// TwinCAT 3 PLC project TcBaseTest
// ProgramVersion: 3.1.4023.0
// libraries:
//   Tc2_Standard, * (Beckhoff Automation GmbH)
//   Tc2_System, * (Beckhoff Automation GmbH)
//   Tc2_Utilities, * (Beckhoff Automation GmbH)
//   Tc3_Module, * (Beckhoff Automation GmbH)
//   TcBase, * (TcBase)
//   TcUnit, * (www.tcunit.org)
// project tree:
//   Action Test/ FB_Action_Test.TcPOU, FB_ActivateAction.TcPOU
//   Collection Test/ FB_ListCapacity_Test.TcPOU, FB_List_proxy.TcPOU, FB_List_Test.TcPOU
//   Invocation Control Test/ FB_InvocationControlTestTask.TcPOU, FB_InvocationControl_Test.TcPOU
//   Object Test/ FB_Object_Test.TcPOU
//   Observer Pattern Test/ FB_ObserverPattern_Test.TcPOU, FB_Observer_LREAL_.TcPOU
//   / PlcTask.TcTTO
//   Programs/ Test.TcPOU
//   State Pattern Test/ FB_StatePattern_Test.TcPOU
//   State Pattern Test/Test Subjects/Dummy State Pattern/ FB_State1.TcPOU, FB_State2.TcPOU, FB_State3.TcPOU, FB_State4.TcPOU, FB_StateMachine1.TcPOU
//   State Pattern Test/Test Subjects/Season State Pattern/ E_Season.TcDUT, FB_Autumn.TcPOU, FB_Default.TcPOU, FB_SeasonBase.TcPOU, FB_SeasonStateMachine.TcPOU, FB_Spring.TcPOU, FB_Summer.TcPOU, FB_Winter.TcPOU, FB_Year.TcPOU, I_SeasonControl.TcIO, I_SeasonState.TcIO
//   Test Objects/ FB_ActionTestObject.TcPOU, FB_TestObject.TcPOU
// real-time tasks:
//   TASK PlcTask: cycle T#10ms, priority 20, ADS port 350

CONFIGURATION TcBaseTest
    RESOURCE PLC ON TwinCAT3
        TASK PlcTask(INTERVAL := T#10ms, PRIORITY := 20);
        PROGRAM Test WITH PlcTask : Test;
    END_RESOURCE
END_CONFIGURATION

// ---- State Pattern Test/Test Subjects/Season State Pattern/E_Season.TcDUT
{attribute 'qualified_only'}
{attribute 'strict'}
{attribute 'to_string'}
TYPE E_Season :
(
    Autumn,
    Winter,
    Spring,
    Summer
);
END_TYPE

// ---- State Pattern Test/Test Subjects/Season State Pattern/I_SeasonControl.TcIO
INTERFACE I_SeasonControl EXTENDS __SYSTEM.IQueryInterface

PROPERTY StateAutumn : I_State
GET
END_GET
END_PROPERTY

PROPERTY StateSpring : I_State
GET
END_GET
END_PROPERTY

PROPERTY StateSummer : I_State
GET
END_GET
END_PROPERTY

PROPERTY StateWinter : I_State
GET
END_GET
END_PROPERTY

END_INTERFACE

// ---- State Pattern Test/Test Subjects/Season State Pattern/I_SeasonState.TcIO
INTERFACE I_SeasonState EXTENDS I_State

PROPERTY bRaining : BOOL
GET
END_GET
END_PROPERTY

PROPERTY bSnowing : BOOL
GET
END_GET
END_PROPERTY

PROPERTY bSunShining : BOOL
GET
END_GET
END_PROPERTY

PROPERTY bWindBlowing : BOOL
GET
END_GET
END_PROPERTY

METHOD ChangeToSummerTyres
VAR_INPUT
END_VAR
END_METHOD

METHOD ChangeToWinterTyres
VAR_INPUT
END_VAR
END_METHOD

PROPERTY eState : E_Season
GET
END_GET
END_PROPERTY

METHOD ABSTRACT NextSeason
VAR_INPUT
END_VAR
END_METHOD

PROPERTY nLeavesState : BYTE
GET
END_GET
END_PROPERTY

PROPERTY nTyresType : BYTE
GET
END_GET
END_PROPERTY

PROPERTY sState : STRING(MAX_STRING_LENGTH)
GET
END_GET
END_PROPERTY

END_INTERFACE

// ---- Programs/Test.TcPOU
PROGRAM Test
VAR
    fbObjectTest: FB_Object_Test;
    fbListTest: FB_List_Test;
    fbListEnsureCapacityTest: FB_ListCapacity_Test;
    fbCallCtrlTest: FB_InvocationControl_Test;
    fbObserverPatternTest: FB_ObserverPattern_Test;
    fbStatePatternTest: FB_StatePattern_Test;
    fbActionTest: FB_Action_Test;
END_VAR

TcUnit.RUN();

END_PROGRAM

// ---- Object Test/FB_Object_Test.TcPOU
{attribute 'reflection'}
FUNCTION_BLOCK FB_Object_Test EXTENDS TcUnit.FB_TestSuite
VAR
    fbPathTester: FB_TestObject;
    _sTestPath: STRING(MAX_STRING_LENGTH) := CONCAT(_sPath, '.fbPathTester');

    {attribute 'instance-path'}
    {attribute 'noinit'}
    _sPath: STRING(MAX_STRING_LENGTH);
END_VAR

TestCompareObjectToSelfExpectTrue();
TestCompareTwoDifferentObjectsExpectFalse();
TestIdentityCorrectness();
TestPathCorrectness();

METHOD PRIVATE TestCompareObjectToSelfExpectTrue
VAR_INST
    fbObject1:      FB_TestObject;
END_VAR
TcUnit.TEST('TestCompareObjectToSelfExpectTrue');

THIS^.AssertTrue(Condition := fbObject1.Equals(fbObject1),
                 Message := 'Failed when comparing two equal objects');

TcUnit.TEST_FINISHED();
END_METHOD

METHOD PRIVATE TestCompareTwoDifferentObjectsExpectFalse
VAR_INST
    fbObject1:      FB_TestObject;
    fbObject2:      FB_TestObject;
END_VAR
TcUnit.TEST('TestCompareTwoDifferentObjectsExpectFalse');

THIS^.AssertFalse(Condition := fbObject1.Equals(fbObject2),
                  Message := 'Failed when comparing two equal objects');

TcUnit.TEST_FINISHED();
END_METHOD

METHOD PRIVATE TestIdentityCorrectness
VAR_INST
    fbObject: FB_TestObject;
END_VAR
TcUnit.TEST('TestIdentityCorrectness');

THIS^.AssertEquals_ULINT(Expected := ADR(fbObject),
                         Actual := fbObject.nIdentity,
                         Message := 'Object indentity is not true');

TcUnit.TEST_FINISHED();
END_METHOD

METHOD PRIVATE TestPathCorrectness
TcUnit.TEST('TestPathCorrectness');

THIS^.AssertEquals_STRING(Expected := THIS^._sTestPath,
                          Actual := THIS^.fbPathTester.sPath,
                          Message := 'Object path is not true');

TcUnit.TEST_FINISHED();
END_METHOD

END_FUNCTION_BLOCK

// ---- Test Objects/FB_TestObject.TcPOU
FUNCTION_BLOCK FB_TestObject EXTENDS FB_Object
VAR_INPUT
END_VAR
VAR_OUTPUT
END_VAR
VAR
    _nTest: INT;
END_VAR

PROPERTY nTest : INT
GET
nTest := THIS^._nTest;
END_GET
SET
THIS^._nTest := nTest;
END_SET
END_PROPERTY

END_FUNCTION_BLOCK

// ---- Collection Test/FB_List_Test.TcPOU
FUNCTION_BLOCK FB_List_Test EXTENDS TcUnit.FB_TestSuite
VAR
END_VAR

TestAdd5DifferentItemsExpectAll5Added();
TestAdd5TimesSameObjectExpectAll5Copies();
TestAddNullInterfaceExpectNothingAdded();
TestClearEmptyListExpectSuccess();
TestClearNonEmptyListExpectSuccess();
TestContainsAddedObjectsExpectSuccess();
TestContainsNullObjectExpectFailure();
TestContainsNullObjectFromEmptyListExpectFailure();
TestCopyToArrayOfCompatibleSizeExpectSuccess();
TestCopyToArrayOfIncompatibleSizeExpectFailure();
TestCopyToArrayWithInvalidIndexExpectFailure();
TestEmptyListMustHaveNoItem();
TestForEachWithActivateActionExpectSuccess();
TestForEachWithCylicTaskActionExpectSuccess();
TestIndexOfItem();
TestInsertIntoEmptyListExpectSuccess();
TestInsertIntoListOfItemsExpectSuccess();
TestLastIndexOfListOfMixedDuplicatesAndUniques();
TestRemoveByIndexAndReAddItemExpectCorrectItemOrder();
TestRemoveByIndexFromEmptyListExpectFailure();
TestRemoveByIndexFromListOf5DifferentItemsExpectSuccess();
TestRemoveByIndexFromListOf5ItemsExpectConsistentContents();
TestRemoveByInvalidIndexFromListOfItemsExpectFailure();
TestRemoveInvalidItemFromListExpectFailure();
TestRemoveValidItemFromListExpectSuccess();
{IF defined (LongTest)}
TestMeasureAddPerformanceWithVeryManyItemsAdded();
{END_IF}

METHOD PRIVATE TestAdd5DifferentItemsExpectAll5Added
VAR_INST
    fbList: FB_List_proxy(0);

    aObject: ARRAY [1..5] OF FB_TestObject;
    ipTmp: I_Object;
    ipCmp: I_Object;
    i: UDINT;
END_VAR
TcUnit.TEST('TestAdd5DifferentItemsExpectAll5Added');

FOR i := 1 TO SIZEOF(aObject)/SIZEOF(aObject[1]) DO
    THIS^.AssertEquals_DINT(Expected := TO_DINT(i - 1),
                            Actual := fbList.AddItem(aObject[i]),
                            Message := 'Failed to add object to list');
END_FOR

THIS^.AssertEquals_UDINT(Expected := SIZEOF(aObject)/SIZEOF(aObject[1]),
                         Actual := fbList.nCount,
                         Message := 'Unexpected number of items added to list');

FOR i := 1 TO SIZEOF(aObject)/SIZEOF(aObject[1]) DO
    ipTmp := fbList.ItemAt(TO_DINT(i - 1));
    ipCmp := aObject[i];
    THIS^.AssertTrue(Condition := ipTmp = ipCmp,
                     Message := CONCAT('Unexpected item at index ', TO_STRING(i)));
END_FOR

TcUnit.TEST_FINISHED();
END_METHOD

METHOD PRIVATE TestAdd5TimesSameObjectExpectAll5Copies
VAR_INST
    fbList: FB_List_proxy(0);

    nTimesToAdd: UDINT;
    fbObject: FB_TestObject;
    ipTmp: I_Object;
    ipCmp: I_Object;
    i: UDINT;
END_VAR
TcUnit.TEST('TestAdd5TimesSameObjectExpectAll5Copies');

nTimesToAdd := 5;

FOR i := 1 TO nTimesToAdd DO
    THIS^.AssertEquals_DINT(Expected := TO_DINT(i - 1),
                            Actual := fbList.AddItem(fbObject),
                            Message := 'Failed to add object to list');
END_FOR

THIS^.AssertEquals_UDINT(Expected := nTimesToAdd,
                         Actual := fbList.nCount,
                         Message := 'Unexpected number of items added to list');

FOR i := 1 TO nTimesToAdd DO
    ipTmp := fbList.ItemAt(TO_DINT(i - 1));
    ipCmp := fbObject;
    THIS^.AssertTrue(Condition := ipTmp = ipCmp,
                     Message := 'Unexpected item added to list');
END_FOR

TcUnit.TEST_FINISHED();
END_METHOD

METHOD PRIVATE TestAddNullInterfaceExpectNothingAdded
VAR_INST
    fbList: FB_List_proxy(0);

    ipTmp: I_Object;
    i: UDINT;
END_VAR
TcUnit.TEST('TestAddNullInterfaceExpectNothingAdded');

FOR i := 1 TO 5 DO
    THIS^.AssertEquals_DINT(Expected := -1,
                            Actual := fbList.AddItem(ipTmp),
                            Message := 'Null item added to list');
END_FOR

THIS^.AssertEquals_UDINT(Expected := 0,
                         Actual := fbList.nCount,
                         Message := 'List has item(s) in it, but it should not');

TcUnit.TEST_FINISHED();
END_METHOD

METHOD PRIVATE TestClearEmptyListExpectSuccess
VAR_INST
    fbList: FB_List_proxy(0);
END_VAR
TcUnit.TEST('TestClearEmptyListExpectSuccess');

fbList.Clear();

THIS^.AssertEquals_UDINT(Expected := 0,
                         Actual := fbList.nCount,
                         Message := 'List should be empty');

TcUnit.TEST_FINISHED();
END_METHOD

METHOD PRIVATE TestClearNonEmptyListExpectSuccess
VAR_INST
    fbList: FB_List_proxy(0);

    aObject: ARRAY [1..5] OF FB_TestObject;
    ipTmp: I_Object;
    i: UDINT;
END_VAR
TcUnit.TEST('TestClearNonEmptyListExpectSuccess');

FOR i := 1 TO SIZEOF(aObject)/SIZEOF(aObject[1]) DO
    fbList.AddItem(aObject[i]);
END_FOR

THIS^.AssertEquals_UDINT(Expected := SIZEOF(aObject)/SIZEOF(aObject[1]),
                         Actual := fbList.nCount,
                         Message := 'Unexpected number of items added to list');

fbList.Clear();

THIS^.AssertEquals_UDINT(Expected := 0,
                         Actual := fbList.nCount,
                         Message := 'List was not correctly cleared');

FOR i := 1 TO SIZEOF(aObject)/SIZEOF(aObject[1]) DO
    ipTmp := fbList.ItemAt(TO_DINT(i));
    THIS^.AssertTrue(Condition := ipTmp = 0,
                     Message := 'List was not correctly cleared');
END_FOR

TcUnit.TEST_FINISHED();
END_METHOD

METHOD PRIVATE TestContainsAddedObjectsExpectSuccess
VAR_INST
    fbList: FB_List_proxy(0);

    aObject: ARRAY [1..5] OF FB_TestObject;

    ipNull: I_Object;
    i: UDINT;
END_VAR
TcUnit.TEST('TestContainsAddedObjectsExpectSuccess');

FOR i := 1 TO SIZEOF(aObject)/SIZEOF(aObject[1]) DO
    fbList.AddItem(aObject[i]);
END_FOR

FOR i := 1 TO SIZEOF(aObject)/SIZEOF(aObject[1]) DO
    THIS^.AssertTrue(Condition := fbList.Contains(aObject[i]),
                     Message := 'List does not contain added item');
END_FOR

THIS^.AssertFalse(Condition := fbList.Contains(ipNull),
                  Message := 'List should not contain null object');

TcUnit.TEST_FINISHED();
END_METHOD

METHOD PRIVATE TestContainsNullObjectExpectFailure
VAR_INST
    fbList: FB_List_proxy(0);

    ipNull: I_Object;
END_VAR
TcUnit.TEST('TestContainsNullObjectExpectFailure');

THIS^.AssertFalse(Condition := fbList.Contains(ipNull),
                  Message := 'List should not contain null object');

TcUnit.TEST_FINISHED();
END_METHOD

METHOD PRIVATE TestContainsNullObjectFromEmptyListExpectFailure
VAR_INST
    fbList: FB_List_proxy(0);

    aObject: ARRAY [1..5] OF FB_TestObject;

    ipNull: I_Object;
    i: UDINT;
END_VAR
TcUnit.TEST('TestContainsNullObjectFromEmptyListExpectFailure');

FOR i := 1 TO SIZEOF(aObject)/SIZEOF(aObject[1]) DO
    fbList.AddItem(aObject[i]);
END_FOR

THIS^.AssertFalse(Condition := fbList.Contains(ipNull),
                  Message := 'List should not contain null object');

TcUnit.TEST_FINISHED();
END_METHOD

METHOD PRIVATE TestCopyToArrayOfCompatibleSizeExpectSuccess
VAR_INST
    fbList: FB_List_proxy(0);
    nObjectCount: UDINT;
    aSrcObject: ARRAY [1..10] OF FB_TestObject;
    aDestObject: ARRAY [1..10] OF I_Object;
    aDestObject2: ARRAY [1..30] OF I_Object;
    i: UDINT;
    ipObject: I_Object;

END_VAR
TcUnit.TEST('TestCopyToArrayOfCompatibleSizeExpectSuccess');

nObjectCount := SIZEOF(aSrcObject)/SIZEOF(aSrcObject[1]);
FOR i := 1 TO nObjectCount DO
    fbList.AddItem(aSrcObject[i]);
END_FOR

// Copy to same size array without offset
THIS^.AssertTrue(Condition := fbList.CopyToArray(aDestObject, 1),
                 Message := 'Failed to copy list to array of same size');

FOR i := 1 TO nObjectCount DO
    ipObject := aSrcObject[i];
    THIS^.AssertTrue(Condition := ipObject = aDestObject[i],
                     Message := 'Expected the same object after in array after copying from list');
END_FOR

// Copy to bigger array with offset
THIS^.AssertTrue(Condition := fbList.CopyToArray(aDestObject2, 14),
                 Message := 'Failed to copy list to array with bigger size');

FOR i := 1 TO nObjectCount DO
    ipObject := aSrcObject[i];
    THIS^.AssertTrue(Condition := ipObject = aDestObject2[i + 13],
                     Message := 'Expected the same object after in array after copying from list');
END_FOR

TcUnit.TEST_FINISHED();
END_METHOD

METHOD PRIVATE TestCopyToArrayOfIncompatibleSizeExpectFailure
VAR_INST
    fbList: FB_List_proxy(0);
    nObjectCount: UDINT;
    aSrcObject: ARRAY [1..10] OF FB_TestObject;
    aDestObject: ARRAY [1..5] OF I_Object;
    i: UDINT;
END_VAR
TcUnit.TEST('TestCopyToArrayOfIncompatibleSizeExpectFailure');

nObjectCount := SIZEOF(aSrcObject)/SIZEOF(aSrcObject[1]);
FOR i := 1 TO nObjectCount DO
    fbList.AddItem(aSrcObject[i]);
END_FOR

THIS^.AssertFalse(Condition := fbList.CopyToArray(aDestObject, 1),
                  Message := 'Failed to copy list to array of same size');

FOR i := 1 TO SIZEOF(aDestObject)/SIZEOF(aDestObject[1]) DO
    THIS^.AssertTrue(Condition := aDestObject[i] = 0,
                     Message := 'Array should be "empty" after copying due to being smaller than list');
END_FOR

TcUnit.TEST_FINISHED();
END_METHOD

METHOD PRIVATE TestCopyToArrayWithInvalidIndexExpectFailure
VAR_INST
    fbList: FB_List_proxy(0);
    nObjectCount: UDINT;
    aSrcObject: ARRAY [1..10] OF FB_TestObject;
    aDestObject: ARRAY [1..10] OF I_Object;
    aDestObject2: ARRAY [1..30] OF I_Object;
    i: UDINT;

END_VAR
TcUnit.TEST('TestCopyToArrayWithInvalidIndexExpectFailure');

nObjectCount := SIZEOF(aSrcObject)/SIZEOF(aSrcObject[1]);
FOR i := 1 TO nObjectCount DO
    fbList.AddItem(aSrcObject[i]);
END_FOR

// Copy to same size array
THIS^.AssertFalse(Condition := fbList.CopyToArray(aDestObject, 2),
                  Message := 'List should not copy items to array using invalid index');

FOR i := 1 TO nObjectCount DO
    THIS^.AssertTrue(Condition := 0 = aDestObject[i],
                     Message := 'Array should be "empty" after copying due to being smaller than list');
END_FOR

// Copy to bigger array
THIS^.AssertFalse(Condition := fbList.CopyToArray(aDestObject2, 22),
                  Message := 'List should not copy items to array using invalid index');

FOR i := 1 TO nObjectCount DO
    THIS^.AssertTrue(Condition := 0 = aDestObject2[i + 13],
                     Message := 'Array should be "empty" after copying due to being smaller than list');
END_FOR

THIS^.AssertFalse(Condition := fbList.CopyToArray(aDestObject2, 0),
                  Message := 'List should not copy items to array using invalid index');

FOR i := 1 TO nObjectCount DO
    THIS^.AssertTrue(Condition := 0 = aDestObject2[i + 13],
                     Message := 'Array should be "empty" after copying due to being smaller than list');
END_FOR

TcUnit.TEST_FINISHED();
END_METHOD

METHOD PRIVATE TestEmptyListMustHaveNoItem
VAR_INST
    fbList:     FB_List_proxy(0);
END_VAR
TcUnit.TEST('TestEmptyListMustHaveNoItem');

THIS^.AssertEquals_UDINT(Expected := 0,
                         Actual := fbList.nCount,
                         Message := 'Empty list must not have any item(s)');

TcUnit.TEST_FINISHED();
END_METHOD

METHOD PRIVATE TestForEachWithActivateActionExpectSuccess
VAR_INST
    i: UDINT;
    fbList: FB_List_proxy(0);
    aObject: ARRAY [1..10] OF FB_ActionTestObject;
    fbActivateObjects: FB_ActivateAction;
END_VAR
TcUnit.TEST('TestForEachWithActivateActionExpectSuccess');

FOR i := 1 TO SIZEOF(aObject)/SIZEOF(aObject[1]) DO
    fbList.AddItem(aObject[i]);
END_FOR

fbList.ForEach(fbActivateObjects.Inputs(TRUE));

FOR i := 1 TO SIZEOF(aObject)/SIZEOF(aObject[1]) DO
     THIS^.AssertTrue(Condition := aObject[1].bIsActivated,
                      Message := 'Failed to activate object(s)');
END_FOR

TcUnit.TEST_FINISHED();
END_METHOD

METHOD PRIVATE TestForEachWithCylicTaskActionExpectSuccess
VAR_INST
    nCyclesToRun: UDINT := 5;
    nCounter: UDINT := 0;
    i: UDINT;
    fbList: FB_List_proxy(0);
    aObject: ARRAY [1..10] OF FB_ActionTestObject;
    fbRunCyclicTask: FB_RunCyclicTasksAction;
END_VAR
TcUnit.TEST('TestForEachWithCylicTaskActionExpectSuccess');

IF nCounter = 0 THEN
    FOR i := 1 TO SIZEOF(aObject)/SIZEOF(aObject[1]) DO
        fbList.AddItem(aObject[i]);
    END_FOR
END_IF

fbList.ForEach(fbRunCyclicTask);
nCounter := nCounter + 1;

IF nCyclesToRun = nCounter THEN
    FOR i := 1 TO SIZEOF(aObject)/SIZEOF(aObject[1]) DO
        THIS^.AssertEquals_UDINT(Expected := nCyclesToRun,
                                 Actual := aObject[i].nCounter,
                                 Message := 'Unexpected counter value of cyclic object');
    END_FOR
    TcUnit.TEST_FINISHED();
END_IF
END_METHOD

METHOD PRIVATE TestIndexOfItem
VAR_INST
    fbList: FB_List_proxy(0);

    aObject: ARRAY [1..10] OF FB_TestObject;
    fbObject1: FB_TestObject;
    fbObject2: FB_TestObject;
    fbObject3: FB_TestObject;

    ipNull: I_Object;
    i: UDINT;
END_VAR
TcUnit.TEST('TestIndexQuerryCorrectness');

FOR i := 1 TO SIZEOF(aObject)/SIZEOF(aObject[1]) DO
    fbList.AddItem(aObject[i]);
END_FOR

FOR i := 1 TO SIZEOF(aObject)/SIZEOF(aObject[1]) DO
    THIS^.AssertEquals_DINT(Expected := TO_DINT(i - 1),
                            Actual := fbList.IndexOfItem(aObject[i]),
                            Message := 'Unexpected index of added item');
END_FOR

fbList.Clear();

FOR i := 1 TO SIZEOF(aObject)/SIZEOF(aObject[1]) DO
    THIS^.AssertEquals_DINT(Expected := -1,
                            Actual := fbList.IndexOfItem(aObject[i]),
                            Message := 'Item still found from list even though it has been cleared');
END_FOR

THIS^.AssertEquals_DINT(Expected := -1,
                        Actual := fbList.IndexOfItem(ipNull),
                        Message := 'Invalid result when querying index of a null item');

fbList.AddItem(fbObject1);
fbList.AddItem(fbObject3);
fbList.AddItem(fbObject1);
fbList.AddItem(fbObject2);
fbList.AddItem(fbObject2);

THIS^.AssertEquals_DINT(Expected := 0,
                        Actual := fbList.IndexOfItem(fbObject1),
                        Message := 'IndexOfItem() should return the index of the first match if there are multiple copies');
THIS^.AssertEquals_DINT(Expected := 1,
                        Actual := fbList.IndexOfItem(fbObject3),
                        Message := 'IndexOfItem() should return the index of the first match if there are multiple copies');
THIS^.AssertEquals_DINT(Expected := 3,
                        Actual := fbList.IndexOfItem(fbObject2),
                        Message := 'IndexOfItem() should return the index of the first match if there are multiple copies');


TcUnit.TEST_FINISHED();
END_METHOD

METHOD PRIVATE TestInsertIntoEmptyListExpectSuccess
VAR_INST
    fbList: FB_List_proxy(0);

    aObject: ARRAY [1..10] OF FB_TestObject;
    aInsPos: ARRAY [1..10] OF DINT;
    ipTmp: I_Object;
    ipCmp: I_Object;

    i: UDINT;
END_VAR
TcUnit.TEST('TestInsertIntoEmptyListExpectSuccess');

FOR i := 1 TO SIZEOF(aObject)/SIZEOF(aObject[1]) DO
    IF i = 4 THEN
        aInsPos[i] := 0;
    ELSIF i = 8 THEN
        aInsPos[i] := 4;;
    ELSIF i = 10 THEN
        aInsPos[i] := 1;
    ELSE
        aInsPos[i] := TO_DINT(i - 1);
    END_IF

    THIS^.AssertTrue(Condition := fbList.Insert(nIdx := aInsPos[i], aObject[i]),
                     Message := 'Could not insert item to list');

    ipTmp := fbList.ItemAt(aInsPos[i]);
    ipCmp := aObject[i];
    THIS^.AssertTrue(Condition := ipTmp = ipCmp,
                     Message := 'Added item is not at the expected index');
END_FOR

THIS^.AssertEquals_UDINT(Expected := SIZEOF(aObject)/SIZEOF(aObject[1]),
                         Actual := fbList.nCount,
                         Message := 'Unexpected number of items inserted to list');

FOR i := 1 TO SIZEOF(aObject)/SIZEOF(aObject[1]) DO
    THIS^.AssertTrue(Condition := fbList.Contains(aObject[i]),
                     Message := 'List does not contain inserted item');
END_FOR

TcUnit.TEST_FINISHED();
END_METHOD

METHOD PRIVATE TestInsertIntoListOfItemsExpectSuccess
VAR_INST
    fbList: FB_List_proxy(0);

    aObject: ARRAY [1..10] OF FB_TestObject;
    aObjectToInsert: ARRAY [1..3] OF FB_TestObject;
    aInsPos: ARRAY [1..3] OF DINT;
    ipTmp: I_Object;
    ipCmp: I_Object;

    i: UDINT;
END_VAR
TcUnit.TEST('TestInsertIntoListOfItemsExpectSuccess');

{region "Insert to head, end, and middle"}
FOR i := 1 TO SIZEOF(aObject)/SIZEOF(aObject[1]) DO
    fbList.AddItem(aObject[i]);
END_FOR

aInsPos[1] := 0;
aInsPos[2] := TO_DINT(fbList.nCount + 1);
aInsPos[3] := 3;

FOR i := 1 TO SIZEOF(aInsPos)/SIZEOF(aInsPos[1]) DO
    THIS^.AssertTrue(Condition := fbList.Insert(aInsPos[i], aObjectToInsert[i]),
                     Message := 'Failed to insert item into list');

    ipTmp := fbList.ItemAt(aInsPos[i]);
    ipCmp := aObjectToInsert[i];
    THIS^.AssertTrue(Condition := ipTmp = ipCmp,
                     Message := 'Added item is not at the expected index');
END_FOR

THIS^.AssertEquals_UDINT(Expected := SIZEOF(aObject)/SIZEOF(aObject[1])
                                     + SIZEOF(aObjectToInsert)/SIZEOF(aObjectToInsert[1]),
                         Actual := fbList.nCount,
                         Message := 'Unexpected number of items inserted to list');

FOR i := 1 TO SIZEOF(aObject)/SIZEOF(aObject[1]) DO
    THIS^.AssertTrue(Condition := fbList.Contains(aObject[i]),
                     Message := 'List does not contain inserted item');
END_FOR

FOR i := 1 TO SIZEOF(aObjectToInsert)/SIZEOF(aObjectToInsert[1]) DO
    THIS^.AssertTrue(Condition := fbList.Contains(aObjectToInsert[i]),
                     Message := 'List does not contain inserted item');
END_FOR
{endregion}

fbList.Clear();

{region "Insert to middle"}
FOR i := 1 TO SIZEOF(aObject)/SIZEOF(aObject[1]) DO
    fbList.AddItem(aObject[i]);
END_FOR

aInsPos[1] := 8;
aInsPos[2] := 5;
aInsPos[3] := 1;

FOR i := 1 TO SIZEOF(aInsPos)/SIZEOF(aInsPos[1]) DO
    THIS^.AssertTrue(Condition := fbList.Insert(aInsPos[i], aObjectToInsert[i]),
                     Message := 'Failed to insert item into list');

    ipTmp := fbList.ItemAt(aInsPos[i]);
    ipCmp := aObjectToInsert[i];
    THIS^.AssertTrue(Condition := ipTmp = ipCmp,
                     Message := 'Added item is not at the expected index');
END_FOR

THIS^.AssertEquals_UDINT(Expected := SIZEOF(aObject)/SIZEOF(aObject[1])
                                     + SIZEOF(aObjectToInsert)/SIZEOF(aObjectToInsert[1]),
                         Actual := fbList.nCount,
                         Message := 'Unexpected number of items inserted to list');

FOR i := 1 TO SIZEOF(aObject)/SIZEOF(aObject[1]) DO
    THIS^.AssertTrue(Condition := fbList.Contains(aObject[i]),
                     Message := 'List does not contain inserted item');
END_FOR

FOR i := 1 TO SIZEOF(aObjectToInsert)/SIZEOF(aObjectToInsert[1]) DO
    THIS^.AssertTrue(Condition := fbList.Contains(aObjectToInsert[i]),
                     Message := 'List does not contain inserted item');
END_FOR
{endregion}

TcUnit.TEST_FINISHED();
END_METHOD

METHOD PRIVATE TestLastIndexOfListOfMixedDuplicatesAndUniques
VAR_INST
    fbList: FB_List_proxy(0);

    aObject: ARRAY [1..5] OF FB_TestObject;
    aAddOrder: ARRAY[1..20] OF I_Object;
    aExpLastIdx: ARRAY [1..5] OF DINT;
    nIdx: UDINT;
    nObjectCount: UDINT;
    nTimesToAdd: UDINT;
    i: UDINT;
    fbRand: DRAND := (Seed := 128);
    sMessage: STRING(255);
END_VAR
TcUnit.TEST('TestLastIndexOfListOfMixedDuplicatesAndUniques');

nObjectCount := SIZEOF(aObject)/SIZEOF(aObject[1]);
nTimesToAdd := SIZEOF(aAddOrder)/SIZEOF(aAddOrder[1]);

FOR i := 1 TO nTimesToAdd DO
    fbRand();
    nIdx := TO_UDINT(fbRand.Num*(nObjectCount - 1)) + 1;
    aAddOrder[i] := aObject[nIdx];

    IF aExpLastIdx[nIdx] < TO_DINT(i) THEN
        aExpLastIdx[nIdx] := TO_DINT(i);
    END_IF
END_FOR

FOR i := 1 TO nTimesToAdd DO
    fbList.AddItem(aAddOrder[i]);
END_FOR

FOR i := 1 TO nObjectCount DO
    sMessage := Tc2_Standard.CONCAT('Unexpected last index of object at idx ', TO_STRING(i));
    THIS^.AssertEquals_DINT(Expected := aExpLastIdx[i] - 1,
                            Actual := fbList.LastIndexOf(aObject[i]),
                            Message := sMessage);
END_FOR

TcUnit.TEST_FINISHED();
END_METHOD

METHOD PRIVATE TestMeasureAddPerformanceWithVeryManyItemsAdded
VAR_INST
    fbList: FB_List_proxy(0);
    fbObject: FB_TestObject;
    fbProfiler: Tc2_Utilities.Profiler;

    nTimesToAdd: UDINT := 100000;
    i: UDINT;
    stProfileData: Tc2_Utilities.PROFILERSTRUCT;
    sMsg: STRING(255);
END_VAR
IF TcUnit.TEST_ORDERED('TestMeasureAddPerformanceWithVeryManyItemsAdded') THEN
    IF nTimesToAdd > 0 THEN
        fbProfiler(START := TRUE, RESET := TRUE);
        FOR i := 1 TO nTimesToAdd DO
            fbList.AddItem(fbObject);
        END_FOR

        THIS^.AssertEquals_UDINT(Expected := TO_UDINT(nTimesToAdd),
                                 Actual := fbList.nCount,
                                 Message := 'Unexpected number of items added to list');

        fbProfiler(START := FALSE);
        stProfileData := fbProfiler.DATA;

        sMsg := 'Took ';
        sMsg := CONCAT(sMsg, TO_STRING(stProfileData.LastExecTime));
        sMsg := CONCAT(sMsg, 'us to add ');
        sMsg := CONCAT(sMsg, TO_STRING(nTimesToAdd));
        sMsg := CONCAT(sMsg, ' item(s) to list. ');
        sMsg := CONCAT(sMsg, 'On average ');
        sMsg := CONCAT(sMsg, TO_STRING(fbProfiler.DATA.AverageExecTime/nTimesToAdd));
        sMsg := CONCAT(sMsg, 'us');
        sMsg := CONCAT(sMsg, ' per item');

        Tc2_System.ADSLOGSTR(msgCtrlMask := Tc2_System.ADSLOG_MSGTYPE_ERROR,
                             msgFmtStr := sMsg,
                             strArg := '');
    END_IF

    TcUnit.TEST_FINISHED();
END_IF
END_METHOD

METHOD PRIVATE TestRemoveByIndexAndReAddItemExpectCorrectItemOrder
VAR_INST
    fbList: FB_List_proxy(0);
    aObject: ARRAY [1..5] OF FB_TestObject;
    aIdx: ARRAY [1..5] OF UDINT
        := [3, 2, 4, 5, 1];
    nArraySize: UDINT;
    i: UDINT;
    j: UDINT;
END_VAR
TcUnit.TEST('TestRemoveByIndexAndReAddItemExpectCorrectItemOrder');
nArraySize := SIZEOF(aObject)/SIZEOF(aObject[1]);

FOR i := 1 TO nArraySize DO
    fbList.AddItem(aObject[i]);
END_FOR

FOR i := 1 TO nArraySize DO
    fbList.RemoveAt(fbList.IndexOfItem(aObject[aIdx[i]]));
    fbList.AddItem(aObject[aIdx[i]]);
END_FOR

FOR i := 1 TO nArraySize DO
    THIS^.AssertTrue(Condition := fbList.ItemAt(TO_DINT(i) - 1).Equals(aObject[aIdx[i]]),
                     Message := CONCAT('Unexpected item found at ', TO_STRING(i - 1)));
END_FOR

TcUnit.TEST_FINISHED();
END_METHOD

METHOD PRIVATE TestRemoveByIndexFromEmptyListExpectFailure
VAR_INST
    fbList: FB_List_proxy(0);

    aIdx: ARRAY[1..10] OF DINT := 
        [0, 1, 2, 3, 4, 5, 6, 7, 8, 9];

    i: UDINT;
END_VAR
TcUnit.TEST('TestRemoveByIndexFromEmptyListExpectFailure');

FOR i := 1 TO SIZEOF(aIdx)/SIZEOF(aIdx[1]) DO
    THIS^.AssertFalse(Condition := fbList.RemoveAt(aIdx[i]),
                      Message := 'Empty list should not have any item to be removed');
END_FOR

TcUnit.TEST_FINISHED();
END_METHOD

METHOD PRIVATE TestRemoveByIndexFromListOf5DifferentItemsExpectSuccess
VAR_INST
    fbList: FB_List_proxy(0);
    aObject: ARRAY [1..5] OF FB_TestObject;

    nArraySize: UDINT;
    i: UDINT;
END_VAR
TcUnit.TEST('TestRemoveItemFromListOf5DifferentItemsExpectSuccess');
nArraySize := SIZEOF(aObject)/SIZEOF(aObject[1]);

// Remove from last to first
FOR i := 1 TO nArraySize DO
    fbList.AddItem(aObject[i]);
END_FOR

FOR i := 1 TO nArraySize DO
    THIS^.AssertTrue(Condition := fbList.RemoveAt(TO_DINT(nArraySize - i)),
                     Message := 'Could not remove added item');

    THIS^.AssertEquals_UDINT(Expected := nArraySize - i,
                             Actual := fbList.nCount,
                             Message := 'Unexpected number of items after removal');
END_FOR

// Remove from first
FOR i := 1 TO nArraySize DO
    fbList.AddItem(aObject[i]);
END_FOR

FOR i := 1 TO nArraySize DO
    THIS^.AssertTrue(Condition := fbList.RemoveAt(0),
                     Message := 'Could not remove added item');

    THIS^.AssertEquals_UDINT(Expected := nArraySize - i,
                             Actual := fbList.nCount,
                             Message := 'Unexpected number of items after removal');
END_FOR

// Remove from middle to first
FOR i := 1 TO nArraySize DO
    fbList.AddItem(aObject[i]);
END_FOR

FOR i := 1 TO nArraySize DO
    THIS^.AssertTrue(Condition := fbList.RemoveAt(MAX(0, 3 - TO_DINT(i))),
                     Message := 'Could not remove added item');

    THIS^.AssertEquals_UDINT(Expected := nArraySize - i,
                             Actual := fbList.nCount,
                             Message := 'Unexpected number of items after removal');
END_FOR

TcUnit.TEST_FINISHED();
END_METHOD

METHOD PRIVATE TestRemoveByIndexFromListOf5ItemsExpectConsistentContents
VAR_INST
    fbList: FB_List_proxy(0);
    aObject: ARRAY [1..5] OF FB_TestObject;
    nArraySize: UDINT;
    i: UDINT;
    j: UDINT;
END_VAR
TcUnit.TEST('TestRemoveByIndexFromListOf5ItemsExpectConsistentContents');
nArraySize := SIZEOF(aObject)/SIZEOF(aObject[1]);

FOR i := 1 TO nArraySize DO
    fbList.AddItem(aObject[i]);
END_FOR

FOR i := 1 TO nArraySize DO
    fbList.RemoveAt(0);

    // After every removal, we check that the content of the list is correct
    IF fbList.nCount > 0 THEN
        FOR j := 0 TO fbList.nCount - 1 DO
            THIS^.AssertTrue(Condition := fbList.ItemAt(TO_DINT(j)).Equals(aObject[i + j + 1]),
                             Message := 'Unexpected list contents after removing item');
        END_FOR
    END_IF
END_FOR

TcUnit.TEST_FINISHED();
END_METHOD

METHOD PRIVATE TestRemoveByInvalidIndexFromListOfItemsExpectFailure
VAR_INST
    fbList: FB_List_proxy(0);

    aIdx: ARRAY[1..10] OF DINT := 
        [-1, 5, 6, 7, 10, -10, -3, -4, -2, 9];
    aObject: ARRAY [1..5] OF FB_TestObject;

    i: UDINT;
END_VAR
TcUnit.TEST('TestRemoveByInvalidIndexFromListOfItemsExpectFailure');

FOR i := 1 TO SIZEOF(aObject)/SIZEOF(aObject[1]) DO
    fbList.AddItem(aObject[i]);
END_FOR

FOR i := 1 TO SIZEOF(aIdx)/SIZEOF(aIdx[1]) DO
    THIS^.AssertFalse(Condition := fbList.RemoveAt(aIdx[i]),
                      Message := 'Removing item with out-of-bound index should not succeed');
END_FOR

THIS^.AssertEquals_UDINT(Expected := 5,
                         Actual := fbList.nCount,
                         Message := 'Item(s) were successfully removed from list with out-of-bound index');

TcUnit.TEST_FINISHED();
END_METHOD

METHOD PRIVATE TestRemoveInvalidItemFromListExpectFailure
VAR_INST
    fbList: FB_List_proxy(0);

    aObject: ARRAY [1..10] OF FB_TestObject;
    ipNull: I_Object;
    fbObject: FB_TestObject;

    i: UDINT;
END_VAR
TcUnit.TEST('TestRemoveInvalidItemFromListExpectFailure');

FOR i := 1 TO SIZEOF(aObject)/SIZEOF(aObject[1]) DO
    fbList.AddItem(aObject[i]);
END_FOR

THIS^.AssertFalse(Condition := fbList.Remove(ipNull),
                  Message := 'Unexpectedly removed a null item');

THIS^.AssertFalse(Condition := fbList.Remove(fbObject),
                  Message := 'List should not be able to remove item it does not contain');

THIS^.AssertEquals_UDINT(Expected := SIZEOF(aObject)/SIZEOF(aObject[1]),
                         Actual := fbList.nCount,
                         Message := 'Unexpected number of items after invalid removal');

FOR i := 1 TO SIZEOF(aObject)/SIZEOF(aObject[1]) DO
    THIS^.AssertTrue(Condition := fbList.Remove(aObject[i]),
                     Message := 'Could not remove added item');

    THIS^.AssertFalse(Condition := fbList.Remove(aObject[i]),
                      Message := 'Removed item was unexpectedly removed twice');

    THIS^.AssertEquals_UDINT(Expected := SIZEOF(aObject)/SIZEOF(aObject[1]) - i,
                             Actual := fbList.nCount,
                             Message := 'Unexpected number of items after removal');
END_FOR

TcUnit.TEST_FINISHED();
END_METHOD

METHOD PRIVATE TestRemoveValidItemFromListExpectSuccess
VAR_INST
    fbList: FB_List_proxy(0);

    aObject: ARRAY [1..10] OF FB_TestObject;

    i: UDINT;
END_VAR
TcUnit.TEST('TestRemoveValidItemFromListExpectSuccess');

FOR i := 1 TO SIZEOF(aObject)/SIZEOF(aObject[1]) DO
    fbList.AddItem(aObject[i]);
END_FOR

FOR i := 1 TO SIZEOF(aObject)/SIZEOF(aObject[1]) DO
    THIS^.AssertTrue(Condition := fbList.Remove(aObject[i]),
                     Message := 'Could not remove added item');

    THIS^.AssertEquals_UDINT(Expected := SIZEOF(aObject)/SIZEOF(aObject[1]) - i,
                             Actual := fbList.nCount,
                             Message := 'Unexpected number of items after removal');
END_FOR

TcUnit.TEST_FINISHED();
END_METHOD

END_FUNCTION_BLOCK

// ---- Collection Test/FB_List_proxy.TcPOU
FUNCTION_BLOCK FB_List_proxy EXTENDS TcBase.FB_List
VAR_INPUT
END_VAR
VAR_OUTPUT
END_VAR
VAR
END_VAR

END_FUNCTION_BLOCK

// ---- Test Objects/FB_ActionTestObject.TcPOU
FUNCTION_BLOCK FB_ActionTestObject EXTENDS TcBase.FB_Object IMPLEMENTS TcBase.I_CyclicTask
VAR
    _nCounter: UDINT;
    _bActivated: BOOL;
END_VAR

METHOD Activate
VAR_INPUT
    bActivate: BOOL;
END_VAR
THIS^._bActivated := bActivate;
END_METHOD

PROPERTY bIsActivated : BOOL
GET
bIsActivated := THIS^._bActivated;
END_GET
END_PROPERTY

PROPERTY nCounter : UDINT
GET
nCounter := THIS^._nCounter;
END_GET
END_PROPERTY

METHOD Run
VAR_INPUT
END_VAR
THIS^._nCounter := THIS^._nCounter + 1;
END_METHOD

END_FUNCTION_BLOCK

// ---- Action Test/FB_ActivateAction.TcPOU
FUNCTION_BLOCK FB_ActivateAction EXTENDS TcBase.FB_Action
VAR
    _bActivated: BOOL;
END_VAR

METHOD  Execute
VAR_INPUT
    ipObject: I_Object;
END_VAR
VAR
    p: POINTER TO FB_ActionTestObject;
END_VAR
__QUERYPOINTER(ipObject, p);

IF p <> 0 THEN
    p^.Activate(THIS^._bActivated);
END_IF
END_METHOD

METHOD Inputs : TcBase.I_Action
VAR_INPUT
    bActivate: BOOL;
END_VAR
Inputs := THIS^;
THIS^._bActivated := bActivate;
END_METHOD

END_FUNCTION_BLOCK

// ---- Collection Test/FB_ListCapacity_Test.TcPOU
FUNCTION_BLOCK FB_ListCapacity_Test EXTENDS TcUnit.FB_TestSuite
VAR_INPUT
END_VAR
VAR_OUTPUT
END_VAR
VAR
END_VAR

TestInitializeCapacityWithNonZeroValuesExpectSuccess();

METHOD PRIVATE TestInitializeCapacityWithNonZeroValuesExpectSuccess
VAR_INST
    aList: ARRAY [1..5] OF FB_List[(4), (10), (20), (100), (1000)];
    aExpected: ARRAY [1..5] OF UDINT := [4, 10, 20, 100, 1000];
    i: UDINT;
END_VAR
TcUnit.TEST('TestInitializeCapacityWithNonZeroValuesExpectSuccess');

FOR i := 1 TO SIZEOF(aList)/SIZEOF(aList[1]) DO
    THIS^.AssertEquals_UDINT(Expected := aExpected[i],
                             Actual := aList[i].nCapacity,
                             Message := 'Unexpected capacity');
END_FOR

TcUnit.TEST_FINISHED();
END_METHOD

END_FUNCTION_BLOCK

// ---- Invocation Control Test/FB_InvocationControl_Test.TcPOU
FUNCTION_BLOCK FB_InvocationControl_Test EXTENDS TcUnit.FB_TestSuite
VAR
    
END_VAR

RunAllTheTimeExpectCalledCyclicallyTrue();
RunAllTheTimeExpectNewInvocationOnce();
RunOnceExpectNewInvocationOnce();
RunOncePerCycleExpectMultipleCallAlwaysFalse();
RunThricePerCycleExpectMultipleCallTrue();

METHOD PRIVATE RunAllTheTimeExpectCalledCyclicallyTrue
VAR_INST
    fbCallCtrl:             FB_InvocationControl;
    fbCallCtrlTestTask:     FB_InvocationControlTestTask;
END_VAR
TcUnit.TEST('RunAllTheTimeExpectCalledCyclicallyTrue');

fbCallCtrlTestTask.SetRunCondition(5).Run();

IF fbCallCtrlTestTask.nCycleCounter = 1 THEN
    THIS^.AssertFalse(Condition := fbCallCtrl.bCalledCyclically,
                      Message := '$'bCalledCyclically$' should be false as Track() has not been called at all');
END_IF

fbCallCtrl.Track();

THIS^.AssertTrue(Condition := fbCallCtrl.bCalledCyclically,
                 Message := '$'bCalledCyclically$' is false, but it should be true');

THIS^.AssertTrue(Condition := fbCallCtrl.bCalledThisCycle,
                 Message := '$'bCalledThisCycle$' is false, but it should be true');

IF fbCallCtrlTestTask.nCycleCounter > 1 THEN
    THIS^.AssertTrue(Condition := fbCallCtrl.bCalledLastCycle,
                     Message := '$'bCalledLastCycle$' is false, but it should be true');
    IF NOT fbCallCtrl.bCalledLastCycle THEN
        ADSLOGSTR(msgCtrlMask := ADSLOG_MSGTYPE_ERROR,
                  msgFmtStr := fbCallCtrl.ToString(),
                  strArg := '');
    END_IF
ELSE
    THIS^.AssertFalse(Condition := fbCallCtrl.bCalledLastCycle,
                      Message := '$'bCalledLastCycle$' should not be true on the first cycle it is called');
END_IF

IF fbCallCtrlTestTask.bDone THEN
    TcUnit.TEST_FINISHED();
END_IF
END_METHOD

METHOD PRIVATE RunAllTheTimeExpectNewInvocationOnce
VAR_INST
    fbCallCtrl:             FB_InvocationControl;
    fbCallCtrlTestTask:     FB_InvocationControlTestTask;
END_VAR
TcUnit.TEST('RunAllTheTimeExpectNewInvocationOnce');

fbCallCtrlTestTask.SetRunCondition(5).Run();

fbCallCtrl.Track();

IF fbCallCtrlTestTask.nCycleCounter = 1 THEN
    THIS^.AssertTrue(Condition := fbCallCtrl.bNewInvocation,
                     Message := '$'bNewInvocation$' is false, but it should be true');
ELSE
    THIS^.Assertfalse(Condition := fbCallCtrl.bNewInvocation,
                      Message := '$'bNewInvocation$' is true, but it should be false');
END_IF

IF fbCallCtrlTestTask.bDone THEN
    TcUnit.TEST_FINISHED();
END_IF
END_METHOD

METHOD PRIVATE RunOnceExpectNewInvocationOnce
VAR_INST
    fbCallCtrl:             FB_InvocationControl;
    fbCallCtrlTestTask:     FB_InvocationControlTestTask;
END_VAR
TcUnit.TEST('RunOnceExpectNewInvocationOnce');

fbCallCtrlTestTask.SetRunCondition(5).Run();

IF fbCallCtrlTestTask.nCycleCounter = 3 THEN
    fbCallCtrl.Track();
    THIS^.AssertTrue(Condition := fbCallCtrl.bNewInvocation,
                     Message := '$'bNewInvocation$' is false, but it should be true');
ELSE
    THIS^.AssertFalse(Condition := fbCallCtrl.bNewInvocation,
                      Message := '$'bNewInvocation$' is trie, but it should be false');
END_IF

IF fbCallCtrlTestTask.bDone THEN
    TcUnit.TEST_FINISHED();
END_IF
END_METHOD

METHOD PRIVATE RunOncePerCycleExpectMultipleCallAlwaysFalse
VAR_INST
    fbCallCtrl:             FB_InvocationControl;
    fbCallCtrlTestTask:     FB_InvocationControlTestTask;
END_VAR
TcUnit.TEST('RunOncePerCycleExpectMultipleCallAlwaysFalse');

fbCallCtrlTestTask.SetRunCondition(5).Run();

THIS^.AssertFalse(Condition := fbCallCtrl.bMultipleCall,
                  Message := '$'bMultipleCall$' is true, but it should be false');

fbCallCtrl.Track();

THIS^.AssertFalse(Condition := fbCallCtrl.bMultipleCall,
                  Message := '$'bMultipleCall$' is true, but it should be false');


IF fbCallCtrlTestTask.bDone THEN
    TcUnit.TEST_FINISHED();
END_IF
END_METHOD

METHOD PRIVATE RunThricePerCycleExpectMultipleCallTrue
VAR_INST
    fbCallCtrl:             FB_InvocationControl;
    fbCallCtrlTestTask:     FB_InvocationControlTestTask;
END_VAR
TcUnit.TEST('RunThricePerCycleExpectMultipleCallTrue');

fbCallCtrlTestTask.SetRunCondition(5).Run();

IF fbCallCtrlTestTask.nCycleCounter > 1 THEN
    THIS^.AssertTrue(Condition := fbCallCtrl.bMultipleCall,
                     Message := '$'bMultipleCall$' is false, but it should be true');
END_IF

fbCallCtrl.Track().Track().Track();

THIS^.AssertTrue(Condition := fbCallCtrl.bMultipleCall,
                 Message := '$'bMultipleCall$' is false, but it should be true');

IF fbCallCtrlTestTask.bDone THEN
    TcUnit.TEST_FINISHED();
END_IF
END_METHOD

END_FUNCTION_BLOCK

// ---- Invocation Control Test/FB_InvocationControlTestTask.TcPOU
FUNCTION_BLOCK FB_InvocationControlTestTask EXTENDS TcBase.FB_Task
VAR CONSTANT
    cDefaultCyclesToRun:        UDINT := 1;
END_VAR
VAR
    _nCyclesToRunIn:            UDINT;

    _nCyclesToRun:              UDINT := 10;
    _nCycleCounter:             UDINT;
END_VAR

PROPERTY nCycleCounter : UDINT
GET
nCycleCounter := THIS^._nCycleCounter;
END_GET
END_PROPERTY

METHOD PROTECTED OnStart
VAR_INPUT
END_VAR
IF THIS^._nCyclesToRunIn > 0 THEN
    THIS^._nCyclesToRun := THIS^._nCyclesToRunIn;
ELSE
    THIS^._nCyclesToRun := THIS^.cDefaultCyclesToRun;
END_IF
END_METHOD

METHOD Restore : I_Restorable
Restore := SUPER^.Restore();

THIS^._nCycleCounter := 0;
END_METHOD

METHOD Run
VAR_INPUT
END_VAR
IF THIS^.Execute() THEN
    THIS^._nCycleCounter := THIS^._nCycleCounter + 1;

    THIS^.DoneWhen(THIS^._nCycleCounter = THIS^._nCyclesToRun);
END_IF
END_METHOD

METHOD SetRunCondition : REFERENCE TO FB_InvocationControlTestTask
VAR_INPUT
    nCyclesToRun:        UDINT; // Number of cycles to run
END_VAR
SetRunCondition REF= THIS^;

THIS^._nCyclesToRunIn := nCyclesToRun;

THIS^.Invoke();
END_METHOD

END_FUNCTION_BLOCK

// ---- Observer Pattern Test/FB_ObserverPattern_Test.TcPOU
FUNCTION_BLOCK FB_ObserverPattern_Test EXTENDS TcUnit.FB_TestSuite
// All observable types implements the same base methods for
// managing the list of observers, hence testing only one type
// of observable is enough. For instance, methods like, `Attach`,
// and `Detach`.
VAR
    fVal: LREAL;
END_VAR

TestAdd5CompatibleObserversExpectAll5();
TestAdd6IncompatibleObserversExpectNone();
TestAddDuplicateObserversExpectFailure();
TestAddNullObserverExpectFailure();
TestClearAllObserversExpectSuccess();
TestCompatibleDataTypesExpectValuesToUpdate();
TestDataTypeConsistencyOfObservables();
TestDataTypeConsistencyOfObservers();
TestDetachAddedObserversExpectSuccess();
TestExternalWithCompatibleDataTypeExpectValueToUpdate();
TestIncompatileDataTypesExpectNoValueChange();
TestNotifyAlwaysUponWriteAccess();
TestNotifyOnlyWhenValueChanged();
TestNotifyUponAttachmentWithObservers();
TestOneObservableToManyObserversExpectAllToUpdateValueAccordingly();

METHOD PRIVATE TestAdd5CompatibleObserversExpectAll5
VAR_INST
    fbObservableReal: FB_Observable_REAL;
    aObserverReal: ARRAY [1..5] OF FB_Observer_REAL;

    i: UDINT;
END_VAR
TcUnit.TEST('TestAdd5CompatibleObserversExpectAll5');

FOR i := 1 TO SIZEOF(aObserverReal)/SIZEOF(aObserverReal[1]) DO
    THIS^.AssertTrue(Condition := fbObservableReal.Attach(aObserverReal[i]),
                     Message := 'Failed to add compatible observer to observable');
END_FOR

THIS^.AssertEquals_UDINT(Expected := 5,
                         Actual := fbObservableReal.nObserverCount,
                         Message := 'Unexpected number of observers attached');

TcUnit.TEST_FINISHED();
END_METHOD

METHOD PRIVATE TestAdd6IncompatibleObserversExpectNone
VAR_INST
    // Test can be less manual with dynamic list
    fbObservableDint: FB_Observable_DINT;
    fbObservableUdint: FB_Observable_UDINT;
    fbObservableUint: FB_Observable_UINT;
    fbObservableReal: FB_Observable_REAL;
    fbObservableLreal: FB_Observable_LREAL;

    fbObserverDint: ARRAY [1..6] OF FB_Observer_DINT;
    fbObserverUdint: ARRAY [1..6] OF FB_Observer_UDINT;
    fbObserverUint: ARRAY [1..6] OF FB_Observer_UINT;
    fbObserverLreal: ARRAY [1..6] OF FB_Observer_LREAL;
    fbObserverReal: ARRAY [1..6] OF FB_Observer_REAL;

    i: UDINT;
END_VAR
TcUnit.TEST('TestAdd6IncompatibleObserversExpectNone');

FOR i := 1 TO SIZEOF(fbObserverUdint)/SIZEOF(fbObserverUdint[1]) DO
    fbObservableDint.Attach(fbObserverUdint[i]);
    fbObservableDint.Attach(fbObserverUint[i]);
    fbObservableDint.Attach(fbObserverLreal[i]);
    fbObservableDint.Attach(fbObserverReal[i]);

    fbObservableUdint.Attach(fbObserverDint[i]);
    fbObservableUdint.Attach(fbObserverUint[i]);
    fbObservableUdint.Attach(fbObserverLreal[i]);
    fbObservableUdint.Attach(fbObserverReal[i]);

    fbObservableUint.Attach(fbObserverDint[i]);
    fbObservableUint.Attach(fbObserverUdint[i]);
    fbObservableUint.Attach(fbObserverLreal[i]);
    fbObservableUint.Attach(fbObserverReal[i]);

    fbObservableLreal.Attach(fbObserverDint[i]);
    fbObservableLreal.Attach(fbObserverUdint[i]);
    fbObservableLreal.Attach(fbObserverUint[i]);
    fbObservableLreal.Attach(fbObserverReal[i]);

    fbObservableReal.Attach(fbObserverDint[i]);
    fbObservableReal.Attach(fbObserverUdint[i]);
    fbObservableReal.Attach(fbObserverUint[i]);
    fbObservableReal.Attach(fbObserverLreal[i]);

END_FOR

THIS^.AssertEquals_UDINT(Expected := 0,
                         Actual := fbObservableDint.nObserverCount,
                         Message := 'Unexpected number of observers attached to observable type DINT');

THIS^.AssertEquals_UDINT(Expected := 0,
                         Actual := fbObservableUdint.nObserverCount,
                         Message := 'Unexpected number of observers attached to observable type UDINT');

THIS^.AssertEquals_UDINT(Expected := 0,
                         Actual := fbObservableUint.nObserverCount,
                         Message := 'Unexpected number of observers attached to observable type UINT');

THIS^.AssertEquals_UDINT(Expected := 0,
                         Actual := fbObservableLreal.nObserverCount,
                         Message := 'Unexpected number of observers attached to observable type LREAL');

THIS^.AssertEquals_UDINT(Expected := 0,
                         Actual := fbObservableReal.nObserverCount,
                         Message := 'Unexpected number of observers attached to observable type REAL');

TcUnit.TEST_FINISHED();
END_METHOD

METHOD PRIVATE TestAddDuplicateObserversExpectFailure
VAR_INST
    fbObservableReal: FB_Observable_REAL;

    fbObserverReal: FB_Observer_REAL;

    i: UDINT;
END_VAR
TcUnit.TEST('TestAddDuplicateObserversExpectFailure');

FOR i := 1 TO 5 DO
    IF i = 1 THEN
        THIS^.AssertTrue(Condition := fbObservableReal.Attach(fbObserverReal),
                         Message := 'Failed to add compatible observer to observable');
    ELSE
        THIS^.AssertFalse(Condition := fbObservableReal.Attach(fbObserverReal),
                          Message := 'Observable should not add duplicate observers');
    END_IF
END_FOR

THIS^.AssertEquals_UDINT(Expected := 1,
                         Actual := fbObservableReal.nObserverCount,
                         Message := 'Unexpected number of observers attached');

TcUnit.TEST_FINISHED();
END_METHOD

METHOD PRIVATE TestAddNullObserverExpectFailure
VAR_INST
    ipNullObs: I_Observer;
    fbObservable: FB_Observable_LREAL;
END_VAR
TcUnit.TEST('TestAddNullObserverExpectFailure');

fbObservable.Attach(ipNullObs);

THIS^.AssertEquals_UDINT(Expected := 0,
                         Actual := fbObservable.nObserverCount,
                         Message := 'Invalid observer added');

TcUnit.TEST_FINISHED();
END_METHOD

METHOD PRIVATE TestClearAllObserversExpectSuccess
VAR_INST
    fbObservableReal: FB_Observable_REAL;
    aObserverReal: ARRAY [1..5] OF FB_Observer_REAL;

    i: UDINT;
END_VAR
TcUnit.TEST('TestClearAllObserversExpectSuccess');

FOR i := 1 TO SIZEOF(aObserverReal)/SIZEOF(aObserverReal[1]) DO
    fbObservableReal.Attach(aObserverReal[i]);
END_FOR

fbObservableReal.ClearAll();

THIS^.AssertEquals_UDINT(Expected := 0,
                         Actual := fbObservableReal.nObserverCount,
                         Message := 'Failed to clear all observers');

TcUnit.TEST_FINISHED();
END_METHOD

METHOD PRIVATE TestCompatibleDataTypesExpectValuesToUpdate
VAR_INST
    fbObservableBool: FB_Observable_BOOL;
    fbObservableByte: FB_Observable_BYTE;
    fbObservableWord: FB_Observable_WORD;
    fbObservableDword: FB_Observable_DWORD;
    fbObservableLword: FB_Observable_LWORD;
    fbObservableSint: FB_Observable_SINT;
    fbObservableUsint: FB_Observable_USINT;
    fbObservableInt: FB_Observable_INT;
    fbObservableUint: FB_Observable_UINT;
    fbObservableDint: FB_Observable_DINT;
    fbObservableUdint: FB_Observable_UDINT;
    fbObservableLint: FB_Observable_LINT;
    fbObservableUlint: FB_Observable_ULINT;
    fbObservableLreal: FB_Observable_LREAL;
    fbObservableReal: FB_Observable_REAL;

    fbObserverBool: FB_Observer_BOOL;
    fbObserverByte: FB_Observer_BYTE;
    fbObserverWord: FB_Observer_WORD;
    fbObserverDword: FB_Observer_DWORD;
    fbObserverLword: FB_Observer_LWORD;
    fbObserverSint: FB_Observer_SINT;
    fbObserverUsint: FB_Observer_USINT;
    fbObserverInt: FB_Observer_INT;
    fbObserverUint: FB_Observer_UINT;
    fbObserverDint: FB_Observer_DINT;
    fbObserverUdint: FB_Observer_UDINT;
    fbObserverLint: FB_Observer_LINT;
    fbObserverUlint: FB_Observer_ULINT;
    fbObserverLreal: FB_Observer_LREAL;
    fbObserverReal: FB_Observer_REAL;

    bVal: BOOL;
    i: UDINT;
END_VAR
TcUnit.TEST('TestCompatibleDataTypesExpectValuesToUpdate');

fbObservableBool.Attach(fbObserverBool);
fbObservableByte.Attach(fbObserverByte);
fbObservableWord.Attach(fbObserverWord);
fbObservableDword.Attach(fbObserverDword);
fbObservableLword.Attach(fbObserverLword);
fbObservableSint.Attach(fbObserverSint);
fbObservableUsint.Attach(fbObserverUsint);
fbObservableUint.Attach(fbObserverUint);
fbObservableInt.Attach(fbObserverInt);
fbObservableDint.Attach(fbObserverDint);
fbObservableUdint.Attach(fbObserverUdint);
fbObservableLint.Attach(fbObserverLint);
fbObservableUlint.Attach(fbObserverUlint);
fbObservableLreal.Attach(fbObserverLreal);
fbObservableReal.Attach(fbObserverReal);

FOR i := 1 TO 10 DO
    bVal := NOT bVal;
    fbObservableBool.bVal := bVal;
    fbObservableByte.nValue8 := TO_BYTE(i);
    fbObservableWord.nValue16 := TO_WORD(i);
    fbObservableDword.nValue32 := TO_DWORD(i);
    fbObservableLword.nValue64 := TO_LWORD(i);
    fbObservableSint.nValue8 := TO_SINT(i);
    fbObservableUsint.nValue8 := TO_USINT(i);
    fbObservableInt.nValue16 := TO_INT(i);
    fbObservableUint.nValue16 := TO_UINT(i);
    fbObservableDint.nValue32 := TO_DINT(i);
    fbObservableUdint.nValue32 := i;
    fbObservableLint.nValue64 := TO_LINT(i);
    fbObservableUlint.nValue64 := TO_ULINT(i);
    fbObservableLreal.fValue64 := TO_LREAL(i);
    fbObservableReal.fValue32 := TO_REAL(i);

    THIS^.AssertEquals_BOOL(Expected := bVal,
                            Actual := fbObserverBool.bValue,
                            Message := 'BOOL observer failed to update value according to observable');
    THIS^.AssertEquals_BYTE(Expected := TO_BYTE(i),
                            Actual := fbObserverByte.nValue8,
                            Message := 'BYTE observer failed to update value according to observable');
    THIS^.AssertEquals_WORD(Expected := TO_WORD(i),
                            Actual := fbObserverWord.nValue16,
                            Message := 'WORD observer failed to update value according to observable');
    THIS^.AssertEquals_DWORD(Expected := TO_DWORD(i),
                             Actual := fbObserverDword.nValue32,
                             Message := 'DWORD observer failed to update value according to observable');
    THIS^.AssertEquals_LWORD(Expected := TO_LWORD(i),
                             Actual := fbObserverLword.nValue64,
                             Message := 'LWORD observer failed to update value according to observable');
    THIS^.AssertEquals_SINT(Expected := TO_SINT(i),
                            Actual := fbObserverSint.nValue8,
                            Message := 'SINT observer failed to update value according to observable');
    THIS^.AssertEquals_USINT(Expected := TO_USINT(i),
                             Actual := fbObserverUsint.nValue8,
                             Message := 'USINT observer failed to update value according to observable');
    THIS^.AssertEquals_INT(Expected := TO_INT(i),
                           Actual := fbObserverInt.nValue16,
                           Message := 'INT observer failed to update value according to observable');
    THIS^.AssertEquals_UINT(Expected := TO_UINT(i),
                            Actual := fbObserverUint.nValue16,
                            Message := 'UINT observer failed to update value according to observable');
    THIS^.AssertEquals_DINT(Expected := TO_DINT(i),
                            Actual := fbObserverDint.nValue32,
                            Message := 'DINT observer failed to update value according to observable');
    THIS^.AssertEquals_UDINT(Expected := i,
                             Actual := fbObserverUdint.nValue32,
                             Message := 'UDINT observer failed to update value according to observable');
    THIS^.AssertEquals_LINT(Expected := TO_LINT(i),
                            Actual := fbObserverLint.nValue64,
                            Message := 'LINT observer failed to update value according to observable');
    THIS^.AssertEquals_LREAL(Expected := TO_LREAL(i),
                             Actual := fbObserverLreal.fValue64,
                             Delta := 0.01,
                             Message := 'LREAL observer failed to update value according to observable');
    THIS^.AssertEquals_REAL(Expected := TO_REAL(i),
                            Actual := fbObserverReal.fValue32,
                            Delta := 0.01,
                            Message := 'REAL observer failed to update value according to observable');
END_FOR

TcUnit.TEST_FINISHED();
END_METHOD

METHOD PRIVATE TestDataTypeConsistencyOfObservables
VAR_INST
    aTypes: ARRAY [1..15] OF __SYSTEM.TYPE_CLASS :=
        [
            __SYSTEM.TYPE_CLASS.TYPE_BOOL,
            __SYSTEM.TYPE_CLASS.TYPE_BYTE,
            __SYSTEM.TYPE_CLASS.TYPE_WORD,
            __SYSTEM.TYPE_CLASS.TYPE_DWORD,
            __SYSTEM.TYPE_CLASS.TYPE_LWORD,
            __SYSTEM.TYPE_CLASS.TYPE_SINT,
            __SYSTEM.TYPE_CLASS.TYPE_USINT,
            __SYSTEM.TYPE_CLASS.TYPE_INT,
            __SYSTEM.TYPE_CLASS.TYPE_UINT,
            __SYSTEM.TYPE_CLASS.TYPE_DINT,
            __SYSTEM.TYPE_CLASS.TYPE_UDINT,
            __SYSTEM.TYPE_CLASS.TYPE_LINT,
            __SYSTEM.TYPE_CLASS.TYPE_ULINT,
            __SYSTEM.TYPE_CLASS.TYPE_LREAL,
            __SYSTEM.TYPE_CLASS.TYPE_REAL
        ];

    fbList: FB_List_proxy(0);
    fbObservableBool: FB_Observable_BOOL;
    fbObservableByte: FB_Observable_BYTE;
    fbObservableWord: FB_Observable_WORD;
    fbObservableDword: FB_Observable_DWORD;
    fbObservableLword: FB_Observable_LWORD;
    fbObservableSint: FB_Observable_SINT;
    fbObservableUsint: FB_Observable_USINT;
    fbObservableInt: FB_Observable_INT;
    fbObservableUint: FB_Observable_UINT;
    fbObservableDint: FB_Observable_DINT;
    fbObservableUdint: FB_Observable_UDINT;
    fbObservableLint: FB_Observable_LINT;
    fbObservableUlint: FB_Observable_ULINT;
    fbObservableLreal: FB_Observable_LREAL;
    fbObservableReal: FB_Observable_REAL;

    ipTmp: I_Observable;
    i: UDINT;
END_VAR
TcUnit.TEST('TestExpectConsistentDataTypeOfObservables');

fbList.AddItem(fbObservableBool);
fbList.AddItem(fbObservableByte);
fbList.AddItem(fbObservableWord);
fbList.AddItem(fbObservableDword);
fbList.AddItem(fbObservableLword);
fbList.AddItem(fbObservableSint);
fbList.AddItem(fbObservableUsint);
fbList.AddItem(fbObservableInt);
fbList.AddItem(fbObservableUint);
fbList.AddItem(fbObservableDint);
fbList.AddItem(fbObservableUdint);
fbList.AddItem(fbObservableLint);
fbList.AddItem(fbObservableUlint);
fbList.AddItem(fbObservableLreal);
fbList.AddItem(fbObservableReal);

FOR i := 1 TO SIZEOF(aTypes)/SIZEOF(aTypes[i]) DO
    __QUERYINTERFACE(fbList.ItemAt(TO_DINT(i - 1)), ipTmp);
    THIS^.AssertEquals_UDINT(Expected := aTypes[i],
                             Actual := ipTmp.nTypeClass,
                             Message := CONCAT('Inconsistent type class for observable tested at index ', TO_STRING(i)));
END_FOR

TcUnit.TEST_FINISHED();
END_METHOD

METHOD PRIVATE TestDataTypeConsistencyOfObservers
VAR_INST
    aTypes: ARRAY [1..15] OF __SYSTEM.TYPE_CLASS :=
        [
            __SYSTEM.TYPE_CLASS.TYPE_BOOL,
            __SYSTEM.TYPE_CLASS.TYPE_BYTE,
            __SYSTEM.TYPE_CLASS.TYPE_WORD,
            __SYSTEM.TYPE_CLASS.TYPE_DWORD,
            __SYSTEM.TYPE_CLASS.TYPE_LWORD,
            __SYSTEM.TYPE_CLASS.TYPE_SINT,
            __SYSTEM.TYPE_CLASS.TYPE_USINT,
            __SYSTEM.TYPE_CLASS.TYPE_INT,
            __SYSTEM.TYPE_CLASS.TYPE_UINT,
            __SYSTEM.TYPE_CLASS.TYPE_DINT,
            __SYSTEM.TYPE_CLASS.TYPE_UDINT,
            __SYSTEM.TYPE_CLASS.TYPE_LINT,
            __SYSTEM.TYPE_CLASS.TYPE_ULINT,
            __SYSTEM.TYPE_CLASS.TYPE_LREAL,
            __SYSTEM.TYPE_CLASS.TYPE_REAL
        ];

    fbList: FB_List_proxy(0);
    fbObserverBool: FB_Observer_BOOL;
    fbObserverByte: FB_Observer_BYTE;
    fbObserverWord: FB_Observer_WORD;
    fbObserverDword: FB_Observer_DWORD;
    fbObserverLword: FB_Observer_LWORD;
    fbObserverSint: FB_Observer_SINT;
    fbObserverUsint: FB_Observer_USINT;
    fbObserverInt: FB_Observer_INT;
    fbObserverUint: FB_Observer_UINT;
    fbObserverDint: FB_Observer_DINT;
    fbObserverUdint: FB_Observer_UDINT;
    fbObserverLint: FB_Observer_LINT;
    fbObserverUlint: FB_Observer_ULINT;
    fbObserverLreal: FB_Observer_LREAL;
    fbObserverReal: FB_Observer_REAL;

    ipTmp: I_Observer;
    i: UDINT;
END_VAR
TcUnit.TEST('TestExpectConsistentDataTypeOfObservers');

fbList.AddItem(fbObserverBool);
fbList.AddItem(fbObserverByte);
fbList.AddItem(fbObserverWord);
fbList.AddItem(fbObserverDword);
fbList.AddItem(fbObserverLword);
fbList.AddItem(fbObserverSint);
fbList.AddItem(fbObserverUsint);
fbList.AddItem(fbObserverInt);
fbList.AddItem(fbObserverUint);
fbList.AddItem(fbObserverDint);
fbList.AddItem(fbObserverUdint);
fbList.AddItem(fbObserverLint);
fbList.AddItem(fbObserverUlint);
fbList.AddItem(fbObserverLreal);
fbList.AddItem(fbObserverReal);

FOR i := 1 TO SIZEOF(aTypes)/SIZEOF(aTypes[i]) DO
    __QUERYINTERFACE(fbList.ItemAt(TO_DINT(i - 1)), ipTmp);
    THIS^.AssertEquals_UDINT(Expected := aTypes[i],
                             Actual := ipTmp.nTypeClass,
                             Message := CONCAT('Inconsistent type class for observable tested at index ', TO_STRING(i)));
END_FOR

TcUnit.TEST_FINISHED();
END_METHOD

METHOD PRIVATE TestDetachAddedObserversExpectSuccess
VAR_INST
    fbObservableReal: FB_Observable_REAL;
    fbObserverReal: ARRAY [1..5] OF FB_Observer_REAL;

    i: UDINT;
END_VAR
TcUnit.TEST('TestDetachAddedObserversExpectSuccess');

FOR i := 1 TO SIZEOF(fbObserverReal)/SIZEOF(fbObserverReal[1]) DO
    fbObservableReal.Attach(fbObserverReal[i]);
END_FOR

FOR i := 1 TO SIZEOF(fbObserverReal)/SIZEOF(fbObserverReal[1]) DO
    THIS^.AssertTrue(Condition := fbObservableReal.Detach(fbObserverReal[i]),
                     Message := 'Failed to deatch added observer');

END_FOR

THIS^.AssertEquals_UDINT(Expected := 0,
                         Actual := fbObservableReal.nObserverCount,
                         Message := 'Unexpected number of observers attached');

TcUnit.TEST_FINISHED();
END_METHOD

METHOD PRIVATE TestExternalWithCompatibleDataTypeExpectValueToUpdate
VAR_INST
    fbObservableLreal: FB_Observable_LREAL;
    fbObserverExt: FB_ObserverExt(THIS^.fVal);
    aTestVal: ARRAY [1..5] OF LREAL :=
        [2.7183, 3.1415, -1, 1.6180, 6.6261];
    i: UDINT;
END_VAR
TcUnit.TEST('TestObserverExternalWithCompatibleDataTypeExpectValueToUpdate');

fbObservableLreal.Attach(fbObserverExt);

FOR i := 1 TO SIZEOF(aTestVal)/SIZEOF(aTestVal[1]) DO
    fbObservableLreal.fValue64 := aTestVal[i];
    THIS^.AssertEquals_LREAL(Expected := aTestVal[i],
                             Actual := THIS^.fVal,
                             Delta := 0.001,
                             Message := 'External observer typed LREAL failed to update value according to observable');
END_FOR

TcUnit.TEST_FINISHED();
END_METHOD

METHOD PRIVATE TestIncompatileDataTypesExpectNoValueChange
VAR_INST
    fbObservableReal: FB_Observable_REAL;

    fbObserverDint: FB_Observer_DINT;
    fbObserverUdint: FB_Observer_UDINT;
    fbObserverUint: FB_Observer_UINT;
    fbObserverLreal: FB_Observer_LREAL;

    i: UDINT;
END_VAR
TcUnit.TEST('TestIncompatileDataTypeObserverAndObservableExpectNoValueChange');

fbObservableReal.Attach(fbObserverDint);
fbObservableReal.Attach(fbObserverUdint);
fbObservableReal.Attach(fbObserverUint);
fbObservableReal.Attach(fbObserverLreal);

FOR i := 1 TO 10 DO
    fbObservableReal.fValue32 := TO_REAL(i);

    THIS^.AssertEquals_DINT(Expected := 0,
                            Actual := fbObserverDint.nValue32,
                            Message := 'DINT observer value is not 0, but it should be 0');

    THIS^.AssertEquals_UDINT(Expected := 0,
                            Actual := fbObserverUdint.nValue32,
                            Message := 'UDINT observer value is not 0, but it should be 0');

    THIS^.AssertEquals_UINT(Expected := 0,
                            Actual := fbObserverUint.nValue16,
                            Message := 'UINT observer value is not 0, but it should be 0');

    THIS^.AssertEquals_LREAL(Expected := 0,
                             Actual := fbObserverLreal.fValue64,
                             Delta := 0.001,
                             Message := 'LREAL observer value is not 0, but it should be 0');
END_FOR

TcUnit.TEST_FINISHED();
END_METHOD

METHOD PRIVATE TestNotifyAlwaysUponWriteAccess
VAR_INST
    fbObservable: FB_Observable_LREAL;
    fbObserver: FB_Observer_LREAL_;

    i: UDINT;
END_VAR
TcUnit.TEST('TestNotifyAlwaysUponWriteAccess');

fbObservable.bNotifyWhenChanged := FALSE;
fbObservable.Attach(fbObserver);

// Expect 1 update already because observable always update its observer upon
// attachment
THIS^.AssertEquals_UDINT(Expected := 1,
                         Actual := fbObserver.nUpdateCounter,
                         Message := 'Unexpected number of updates to observer');

FOR i := 1 TO 5 DO
    fbObservable.fValue64 := 1.0;
END_FOR

THIS^.AssertEquals_UDINT(Expected := 6,
                         Actual := fbObserver.nUpdateCounter,
                         Message := 'Unexpected number of updates to observer');

TcUnit.TEST_FINISHED();
END_METHOD

METHOD PRIVATE TestNotifyOnlyWhenValueChanged
VAR_INST
    fbObservable: FB_Observable_LREAL;
    fbObserver: FB_Observer_LREAL_;
    aVal: ARRAY [1..5] OF LREAL :=
        [2.7183, 3.1415, -1, 1.6180, 6.6261];

    i: UDINT;
    j: UDINT;
END_VAR
TcUnit.TEST('TestNotifyOnlyWhenValueChanged');

fbObservable.bNotifyWhenChanged := TRUE;
fbObservable.Attach(fbObserver);

// Expect 1 update already because observable always update its observer upon
// attachment
THIS^.AssertEquals_UDINT(Expected := 1,
                         Actual := fbObserver.nUpdateCounter,
                         Message := 'Unexpected number of updates to observer');

FOR i := 1 TO SIZEOF(aVal)/SIZEOF(aVal[1]) DO
    FOR j := 1 TO 5 DO
        fbObservable.fValue64 := aVal[i];
    END_FOR

    THIS^.AssertEquals_UDINT(Expected := i + 1,
                             Actual := fbObserver.nUpdateCounter,
                             Message := 'Unexpected number of updates to observer');
END_FOR


TcUnit.TEST_FINISHED();
END_METHOD

METHOD PRIVATE TestNotifyUponAttachmentWithObservers
VAR_INST
    fbObservable: FB_Observable_LREAL;
    aObserver: ARRAY [1..5] OF FB_Observer_LREAL_;

    i: UDINT;
END_VAR
TcUnit.TEST('TestNotifyUponAttachmentWithObservers');

fbObservable.fValue64 := 100.0;

FOR i := 1 TO SIZEOF(aObserver)/SIZEOF(aObserver[1]) DO
    fbObservable.Attach(aObserver[i]);
END_FOR

FOR i := 1 TO SIZEOF(aObserver)/SIZEOF(aObserver[1]) DO
    THIS^.AssertEquals_LREAL(Expected := fbObservable.fValue64,
                             Actual := aObserver[i].fValue64,
                             Delta := 0.01,
                             Message := 'Observer$'s value is not matching its observable upon attachment');
    THIS^.AssertEquals_UDINT(Expected := 1,
                             Actual := aObserver[i].nUpdateCounter,
                             Message := 'Unexpected number of updates to observer');
END_FOR

TcUnit.TEST_FINISHED();
END_METHOD

METHOD PRIVATE TestOneObservableToManyObserversExpectAllToUpdateValueAccordingly
VAR_INST
    fbObservableLreal: FB_Observable_LREAL;
    aObservers: ARRAY [1..5] OF FB_Observer_LREAL;
    aTestVal: ARRAY [1..5] OF LREAL :=
        [2.7183, 3.1415, -1, 1.6180, 6.6261];
    i: UDINT;
    j: UDINT;
END_VAR
TcUnit.TEST('TestOneObservableToManyObserversExpectAllToUpdateValueAccordingly');

FOR i := 1 TO SIZEOF(aObservers)/SIZEOF(aObservers[1]) DO
    fbObservableLreal.Attach(aObservers[i]);
END_FOR

FOR i := 1 TO SIZEOF(aTestVal)/SIZEOF(aTestVal[1]) DO
    fbObservableLreal.fValue64 := aTestVal[i];
    FOR j := 1 TO SIZEOF(aObservers)/SIZEOF(aObservers[1]) DO
        THIS^.AssertEquals_LREAL(Expected := aTestVal[i],
                         Actual := aObservers[j].fValue64,
                         Delta := 0.001,
                         Message := ' typed LREAL failed to update value according to observable');
    END_FOR
END_FOR

TcUnit.TEST_FINISHED();
END_METHOD

END_FUNCTION_BLOCK

// ---- Observer Pattern Test/FB_Observer_LREAL_.TcPOU
FUNCTION_BLOCK FB_Observer_LREAL_ EXTENDS TcBase.FB_Observer_LREAL
VAR_INPUT
END_VAR
VAR_OUTPUT
END_VAR
VAR
END_VAR

PROPERTY nUpdateCounter : UDINT
GET
nUpdateCounter := THIS^._nUpdateCounter;
END_GET
END_PROPERTY

END_FUNCTION_BLOCK

// ---- State Pattern Test/FB_StatePattern_Test.TcPOU
FUNCTION_BLOCK FB_StatePattern_Test EXTENDS TcUnit.FB_TestSuite IMPLEMENTS TcBase.I_Object
VAR
    _ipSelf:            I_Object;

    fbStateMachine1:    FB_StateMachine1;
    fbState11:          FB_State1(0);
    fbState12:          FB_State2(0);
    fbState13:          FB_State3(0);
    fbState14:          FB_State4(0);

    fbStateMachine2:    FB_StateMachine1;
    fbState21:          FB_State1(THIS^.fbStateMachine2);
    fbState22:          FB_State2(THIS^.fbStateMachine2);
    fbState23:          FB_State3(THIS^.fbStateMachine2);
    fbState24:          FB_State4(THIS^.fbStateMachine2);

    fbYear:             FB_Year;
END_VAR

TestAdd4StatesByInitializationExpectSuccess();
TestAdd4StatesManuallyExpectSuccess();
TestClearAllStatesExpectSuccess();
TestSeasonStateMachineAllSeasons();

METHOD Equals : BOOL
VAR_INPUT
    ipObject:       TcBase.I_Object;
END_VAR
Equals := ipObject = THIS^._ipSelf;
END_METHOD

PROPERTY ipContext : TcBase.I_Context
GET
ipContext := 0;
END_GET
END_PROPERTY

PROPERTY nIdentity : ULINT
GET
nIdentity := ADR(THIS^);
END_GET
END_PROPERTY

PROPERTY sPath : STRING(MAX_STRING_LENGTH)
GET
sPath := '';
END_GET
END_PROPERTY

METHOD PRIVATE TestAdd4StatesByInitializationExpectSuccess
TcUnit.TEST('TestAdd4StatesByInitializationExpectSuccess');

THIS^.AssertEquals_UDINT(Expected := 4,
                         Actual := THIS^.fbStateMachine2.nStateCount,
                         Message := 'Unexpected number of states added to state machine');
THIS^.AssertTrue(Condition := THIS^.fbStateMachine2.Contains(THIS^.fbState21),
                 Message := 'State machine does not contain added state fbState5');
THIS^.AssertTrue(Condition := THIS^.fbStateMachine2.Contains(THIS^.fbState22),
                 Message := 'State machine does not contain added state fbState6');
THIS^.AssertTrue(Condition := THIS^.fbStateMachine2.Contains(THIS^.fbState23),
                 Message := 'State machine does not contain added state fbState7');
THIS^.AssertTrue(Condition := THIS^.fbStateMachine2.Contains(THIS^.fbState24),
                 Message := 'State machine does not contain added state fbState8');

THIS^.AssertTrue(Condition := THIS^.fbState21.ipStateMachine.Equals(THIS^.fbStateMachine2),
                 Message := 'State fbState5 does not point to the correct state machine');
THIS^.AssertTrue(Condition := THIS^.fbState22.ipStateMachine.Equals(THIS^.fbStateMachine2),
                 Message := 'State fbState6 does not point to the correct state machine');
THIS^.AssertTrue(Condition := THIS^.fbState23.ipStateMachine.Equals(THIS^.fbStateMachine2),
                 Message := 'State fbState7 does not point to the correct state machine');
THIS^.AssertTrue(Condition := THIS^.fbState24.ipStateMachine.Equals(THIS^.fbStateMachine2),
                 Message := 'State fbState8 does not point to the correct state machine');


TcUnit.TEST_FINISHED();
END_METHOD

METHOD PRIVATE TestAdd4StatesManuallyExpectSuccess
TcUnit.TEST_ORDERED('TestAdd4StatesManuallyExpectSuccess');

THIS^.AssertTrue(Condition := THIS^.fbStateMachine1.AddState(THIS^.fbState11),
                 Message := 'Failed to add fbState1 to fbStateMachine');
THIS^.AssertFalse(Condition := THIS^.fbStateMachine1.AddState(THIS^.fbState11),
                  Message := 'fbState1 has already been added to fbStateMachine');
THIS^.AssertEquals_UDINT(Expected := 1,
                         Actual := THIS^.fbStateMachine1.nStateCount,
                         Message := 'Unexpected number of states added to state machine');
THIS^.AssertTrue(Condition := THIS^.fbState11.ipStateMachine.Equals(THIS^.fbStateMachine1),
                 Message := 'State fbState1 does not point to the correct state machine');

THIS^.AssertTrue(Condition := THIS^.fbStateMachine1.AddState(THIS^.fbState12),
                 Message := 'Failed to add fbState2 to fbStateMachine');
THIS^.AssertFalse(Condition := THIS^.fbStateMachine1.AddState(THIS^.fbState12),
                  Message := 'fbState2 has already been added to fbStateMachine');
THIS^.AssertEquals_UDINT(Expected := 2,
                         Actual := THIS^.fbStateMachine1.nStateCount,
                         Message := 'Unexpected number of states added to state machine');
THIS^.AssertTrue(Condition := THIS^.fbState12.ipStateMachine.Equals(THIS^.fbStateMachine1),
                 Message := 'State fbState2 does not point to the correct state machine');

THIS^.AssertTrue(Condition := THIS^.fbStateMachine1.AddState(THIS^.fbState13),
                 Message := 'Failed to add fbState3 to fbStateMachine');
THIS^.AssertFalse(Condition := THIS^.fbStateMachine1.AddState(THIS^.fbState13),
                  Message := 'fbState2 has already been added to fbStateMachine');
THIS^.AssertEquals_UDINT(Expected := 3,
                         Actual := THIS^.fbStateMachine1.nStateCount,
                         Message := 'Unexpected number of states added to state machine');
THIS^.AssertTrue(Condition := THIS^.fbState13.ipStateMachine.Equals(THIS^.fbStateMachine1),
                 Message := 'State fbState3 does not point to the correct state machine');

THIS^.AssertTrue(Condition := THIS^.fbStateMachine1.AddState(THIS^.fbState14),
                 Message := 'Failed to add fbState4 to fbStateMachine');
THIS^.AssertFalse(Condition := THIS^.fbStateMachine1.AddState(THIS^.fbState14),
                  Message := 'fbState2 has already been added to fbStateMachine');
THIS^.AssertEquals_UDINT(Expected := 4,
                         Actual := THIS^.fbStateMachine1.nStateCount,
                         Message := 'Unexpected number of states added to state machine');
THIS^.AssertTrue(Condition := THIS^.fbState14.ipStateMachine.Equals(THIS^.fbStateMachine1),
                 Message := 'State fbState4 does not point to the correct state machine');

THIS^.AssertTrue(Condition := THIS^.fbStateMachine1.Contains(THIS^.fbState11),
                 Message := 'State machine does not contain added state fbState1');
THIS^.AssertTrue(Condition := THIS^.fbStateMachine1.Contains(THIS^.fbState12),
                 Message := 'State machine does not contain added state fbState2');
THIS^.AssertTrue(Condition := THIS^.fbStateMachine1.Contains(THIS^.fbState13),
                 Message := 'State machine does not contain added state fbState3');
THIS^.AssertTrue(Condition := THIS^.fbStateMachine1.Contains(THIS^.fbState14),
                 Message := 'State machine does not contain added state fbState4');

TcUnit.TEST_FINISHED();
END_METHOD

METHOD PRIVATE TestClearAllStatesExpectSuccess
VAR_INPUT
END_VAR
TcUnit.TEST_ORDERED('TestClearAllStatesExpectSuccess');

THIS^.fbStateMachine1.ClearStates();

THIS^.AssertEquals_UDINT(Expected := 0,
                         Actual := THIS^.fbStateMachine1.nStateCount,
                         Message := 'State machine did not clear all states correctly');

THIS^.AssertFalse(Condition := THIS^.fbStateMachine1.Contains(THIS^.fbState11),
                  Message := 'Cleared state should not be in state machine');
THIS^.AssertFalse(Condition := THIS^.fbStateMachine1.Contains(THIS^.fbState12),
                  Message := 'Cleared state should not be in state machine');
THIS^.AssertFalse(Condition := THIS^.fbStateMachine1.Contains(THIS^.fbState13),
                  Message := 'Cleared state should not be in state machine');
THIS^.AssertFalse(Condition := THIS^.fbStateMachine1.Contains(THIS^.fbState14),
                  Message := 'Cleared state should not be in state machine');

TcUnit.TEST_FINISHED();
END_METHOD

METHOD PRIVATE TestSeasonStateMachineAllSeasons
VAR_INPUT
END_VAR
TcUnit.TEST('TestSeasonStateMachineAllSeasons');

THIS^.fbYear.Run();

// Summer
THIS^.AssertEquals_BYTE(Expected := 1,
                        Actual := THIS^.fbYear.CurrentState().nTyresType,
                        Message := 'Tyres initialization is incorrect for Summer');
THIS^.AssertTrue(Condition := THIS^.fbYear.CurrentState().Equals(THIS^.fbYear.StateSummer),
                 Message := 'Expected Summer to be the starting season');
THIS^.AssertTrue(Condition := THIS^.fbYear.CurrentState().bSunShining,
                 Message := 'Expected the sun to shine during Summer');
THIS^.AssertEquals_BYTE(Expected := 1,
                        Actual := THIS^.fbYear.CurrentState().nLeavesState,
                        Message := 'Expected the color of the leaves to be green');
THIS^.fbYear.ChangeToWinterTyres();
THIS^.AssertEquals_BYTE(Expected := 1,
                        Actual := THIS^.fbYear.CurrentState().nTyresType,
                        Message := 'Must not be able to put winter tyres on during Summer');

// Autumn
THIS^.fbYear.NextSeason();
THIS^.AssertTrue(Condition := THIS^.fbYear.CurrentState().Equals(THIS^.fbYear.StateAutumn),
                 Message := 'Expected Autumn to be after Summer');
THIS^.AssertTrue(Condition := THIS^.fbYear.CurrentState().bWindBlowing,
                 Message := 'Expected the wind to blow during Autumn');
THIS^.AssertEquals_BYTE(Expected := 2,
                        Actual := THIS^.fbYear.CurrentState().nLeavesState,
                        Message := 'Expected the color of the leaves to be (changing to) yellow/orange/red');
THIS^.fbYear.ChangeToWinterTyres();
THIS^.AssertEquals_BYTE(Expected := 1,
                        Actual := THIS^.fbYear.CurrentState().nTyresType,
                        Message := 'Must not be able to put winter tyres on during Autumn');

// Winter
THIS^.fbYear.NextSeason();
THIS^.AssertTrue(Condition := THIS^.fbYear.CurrentState().Equals(THIS^.fbYear.StateWinter),
                 Message := 'Expected Winter to be after Autumn');
THIS^.AssertTrue(Condition := THIS^.fbYear.CurrentState().bSnowing,
                 Message := 'Expected snow during Winter');
THIS^.AssertEquals_BYTE(Expected := 0,
                        Actual := THIS^.fbYear.CurrentState().nLeavesState,
                        Message := 'Expected (some) leaves to have been fallen off');
THIS^.fbYear.ChangeToWinterTyres();
THIS^.AssertEquals_BYTE(Expected := 0,
                        Actual := THIS^.fbYear.CurrentState().nTyresType,
                        Message := 'Failed to be able to put winter tyres on');

// Spring
THIS^.fbYear.NextSeason();
THIS^.AssertTrue(Condition := THIS^.fbYear.CurrentState().Equals(THIS^.fbYear.StateSpring),
                 Message := 'Expected Spring to be after Winter');
THIS^.AssertTrue(Condition := THIS^.fbYear.CurrentState().bRaining,
                 Message := 'Expected rain during Spring');
THIS^.AssertEquals_BYTE(Expected := 1,
                        Actual := THIS^.fbYear.CurrentState().nLeavesState,
                        Message := 'Expected the color of the leaves to be green');
THIS^.fbYear.ChangeToSummerTyres();
THIS^.AssertEquals_BYTE(Expected := 1,
                        Actual := THIS^.fbYear.CurrentState().nTyresType,
                        Message := 'Failed to be able to put summer tyres on');

TcUnit.TEST_FINISHED();
END_METHOD

END_FUNCTION_BLOCK

// ---- State Pattern Test/Test Subjects/Dummy State Pattern/FB_StateMachine1.TcPOU
FUNCTION_BLOCK FB_StateMachine1 EXTENDS FB_StateMachine
VAR_INPUT
END_VAR
VAR_OUTPUT
END_VAR
VAR
END_VAR

END_FUNCTION_BLOCK

// ---- State Pattern Test/Test Subjects/Dummy State Pattern/FB_State1.TcPOU
FUNCTION_BLOCK FB_State1 EXTENDS FB_State
VAR_INPUT
END_VAR
VAR_OUTPUT
END_VAR
VAR
END_VAR

END_FUNCTION_BLOCK

// ---- State Pattern Test/Test Subjects/Dummy State Pattern/FB_State2.TcPOU
FUNCTION_BLOCK FB_State2 EXTENDS FB_State
VAR_INPUT
END_VAR
VAR_OUTPUT
END_VAR
VAR
END_VAR

END_FUNCTION_BLOCK

// ---- State Pattern Test/Test Subjects/Dummy State Pattern/FB_State3.TcPOU
FUNCTION_BLOCK FB_State3 EXTENDS FB_State
VAR_INPUT
END_VAR
VAR_OUTPUT
END_VAR
VAR
END_VAR

END_FUNCTION_BLOCK

// ---- State Pattern Test/Test Subjects/Dummy State Pattern/FB_State4.TcPOU
FUNCTION_BLOCK FB_State4 EXTENDS FB_State
VAR_INPUT
END_VAR
VAR_OUTPUT
END_VAR
VAR
END_VAR

END_FUNCTION_BLOCK

// ---- State Pattern Test/Test Subjects/Season State Pattern/FB_Year.TcPOU
FUNCTION_BLOCK FB_Year EXTENDS FB_Object IMPLEMENTS I_SeasonControl, I_CyclicTask
VAR
    fbSeasonStateMachine:   FB_SeasonStateMachine;
    fbWinter:               FB_Winter(THIS^.fbSeasonStateMachine, THIS^);
    fbSpring:               FB_Spring(THIS^.fbSeasonStateMachine, THIS^);
    fbSummer:               FB_Summer(THIS^.fbSeasonStateMachine, THIS^);
    fbAutumn:               FB_Autumn(THIS^.fbSeasonStateMachine, THIS^);

    nCounter:               UDINT;
    nModVal:                UDINT := 500;
END_VAR

METHOD ChangeToSummerTyres
VAR_INPUT
END_VAR
THIS^.CurrentState().ChangeToSummerTyres();
END_METHOD

METHOD ChangeToWinterTyres
VAR_INPUT
END_VAR
THIS^.CurrentState().ChangeToWinterTyres();
END_METHOD

METHOD CurrentState : I_SeasonState
__QUERYINTERFACE(THIS^.fbSeasonStateMachine.ipState, CurrentState);
END_METHOD

METHOD FB_init : BOOL
VAR_INPUT
    bInitRetains:           BOOL; // if TRUE, the retain variables are initialized (warm start / cold start)
    bInCopyCode:            BOOL;  // if TRUE, the instance afterwards gets moved into the copy code (online change)
END_VAR
THIS^.fbSeasonStateMachine.SetState(THIS^.StateSummer);
THIS^.CurrentState().ChangeToSummerTyres();
END_METHOD

METHOD NextSeason
VAR_INPUT
END_VAR
THIS^.fbSeasonStateMachine.NextSeason();
END_METHOD

METHOD Run
VAR_INPUT
END_VAR
THIS^.nCounter := THIS^.nCounter + 1;
THIS^.fbSeasonStateMachine.Run();
END_METHOD

PROPERTY StateAutumn : I_State
GET
StateAutumn := THIS^.fbAutumn;
END_GET
END_PROPERTY

PROPERTY StateSpring : I_State
GET
StateSpring := THIS^.fbSpring;
END_GET
END_PROPERTY

PROPERTY StateSummer : I_State
GET
StateSummer := THIS^.fbSummer;
END_GET
END_PROPERTY

PROPERTY StateWinter : I_State
GET
StateWinter := THIS^.fbWinter;
END_GET
END_PROPERTY

END_FUNCTION_BLOCK

// ---- State Pattern Test/Test Subjects/Season State Pattern/FB_SeasonStateMachine.TcPOU
FUNCTION_BLOCK FB_SeasonStateMachine EXTENDS FB_StateMachine
VAR
    fbDefaultState:     FB_Default(THIS^, THIS^);
END_VAR

METHOD CurrentSeason : I_SeasonState
VAR_INPUT
END_VAR
__QUERYINTERFACE(THIS^.ipState, CurrentSeason);

IF CurrentSeason = 0 THEN
    CurrentSeason := THIS^.fbDefaultState;
END_IF
END_METHOD

METHOD NextSeason
VAR_INPUT
END_VAR
THIS^.CurrentSeason().NextSeason();
END_METHOD

PROPERTY StateDefault : I_SeasonState
GET
StateDefault := THIS^.fbDefaultState;
END_GET
END_PROPERTY

END_FUNCTION_BLOCK

// ---- State Pattern Test/Test Subjects/Season State Pattern/FB_Default.TcPOU
FUNCTION_BLOCK FB_Default EXTENDS FB_SeasonBase
VAR
END_VAR

METHOD  NextSeason
VAR_INST
    fbCallCtrl:     FB_InvocationControl;
END_VAR
IF fbCallCtrl.Track().bNewInvocation THEN
    Tc2_System.ADSLOGSTR(msgCtrlMask := THIS^._nLogLevel,
                         msgFmtStr := 'Current state for %s is not initialized!',
                         strArg := THIS^.sPath);
END_IF

IF THIS^.ipStateMachine <> 0 THEN
    THIS^.ipStateMachine.SetState(THIS^);
END_IF
END_METHOD

END_FUNCTION_BLOCK

// ---- State Pattern Test/Test Subjects/Season State Pattern/FB_SeasonBase.TcPOU
FUNCTION_BLOCK ABSTRACT FB_SeasonBase EXTENDS FB_State IMPLEMENTS I_SeasonState
VAR
    _ipWeatherCtrl:     I_SeasonControl;
    _eState:            E_Season;
END_VAR
VAR_STAT
    _bWindBlowing:      BOOL;
    _bRaining:          BOOL;
    _bSunShining:       BOOL;
    _bSnowing:          BOOL;
    _nTyresType:        BYTE; // 0: winter, 1: summer/all season
    _nLeavesState:      BYTE; // 0: no leave, 1: green leaves, 2: yellow/orange/red leaves
    _nCounter:          UDINT;
    _nModVal:           UDINT := 500;
    _nLogLevel:         DWORD := Tc2_System.ADSLOG_MSGTYPE_WARN;
END_VAR

PROPERTY FINAL bRaining : BOOL
GET
bRaining := THIS^._bRaining;
END_GET
END_PROPERTY

PROPERTY FINAL bSnowing : BOOL
GET
bSnowing := THIS^._bSnowing;
END_GET
END_PROPERTY

PROPERTY FINAL bSunShining : BOOL
GET
bSunShining := THIS^._bSunShining;
END_GET
END_PROPERTY

PROPERTY FINAL bWindBlowing : BOOL
GET
bWindBlowing := THIS^._bWindBlowing;
END_GET
END_PROPERTY

METHOD ChangeToSummerTyres
VAR_INPUT
END_VAR
END_METHOD

METHOD ChangeToWinterTyres
VAR_INPUT
END_VAR
END_METHOD

PROPERTY FINAL eState : E_Season
GET
eState := THIS^._eState;
END_GET
END_PROPERTY

METHOD FB_init : BOOL
VAR_INPUT
    bInitRetains:           BOOL; // if TRUE, the retain variables are initialized (warm start / cold start)
    bInCopyCode:            BOOL;  // if TRUE, the instance afterwards gets moved into the copy code (online change)
    ipStateMachine:         I_StateMachine;
    ipParentObject:         I_Object;
END_VAR
__QUERYINTERFACE(ipParentObject, THIS^._ipWeatherCtrl);
END_METHOD

PROPERTY ipSeasonCtrl : I_SeasonControl
GET
ipSeasonCtrl := THIS^._ipWeatherCtrl;
END_GET
END_PROPERTY

METHOD ABSTRACT NextSeason
VAR_INPUT
END_VAR
END_METHOD

PROPERTY FINAL nLeavesState : BYTE
GET
nLeavesState := THIS^._nLeavesState;
END_GET
END_PROPERTY

PROPERTY FINAL nTyresType : BYTE
GET
nTyresType := THIS^._nTyresType;
END_GET
END_PROPERTY

METHOD OnEntry
VAR
    sTmp:       STRING(MAX_STRING_LENGTH);
END_VAR
sTmp := CONCAT(THIS^.sState, ' here we go!');

Tc2_System.ADSLOGSTR(msgCtrlMask := THIS^._nLogLevel,
                     msgFmtStr := sTmp,
                     strArg := '');

IF THIS^.bWindBlowing THEN
    Tc2_System.ADSLOGSTR(msgCtrlMask := THIS^._nLogLevel,
                         msgFmtStr := 'The wind is blowing',
                         strArg := '');
END_IF

IF THIS^.bRaining THEN
    Tc2_System.ADSLOGSTR(msgCtrlMask := THIS^._nLogLevel,
                         msgFmtStr := 'It$'s raining dogs and cats',
                         strArg := '');
END_IF

IF THIS^.bSunShining THEN
    Tc2_System.ADSLOGSTR(msgCtrlMask := THIS^._nLogLevel,
                         msgFmtStr := 'Aurinko paistaa',
                         strArg := '');
END_IF

IF THIS^.bSnowing THEN
    Tc2_System.ADSLOGSTR(msgCtrlMask := THIS^._nLogLevel,
                         msgFmtStr := 'Sataa lunta',
                         strArg := '');
END_IF
END_METHOD

METHOD OnExit
VAR
    sTmp:       STRING(MAX_STRING_LENGTH);
END_VAR
sTmp := CONCAT('Good bye ', THIS^.sState);

Tc2_System.ADSLOGSTR(msgCtrlMask := THIS^._nLogLevel,
                     msgFmtStr := sTmp,
                     strArg := '');
END_METHOD

METHOD Run
VAR_INPUT
END_VAR
THIS^._nCounter := THIS^._nCounter + 1;
END_METHOD

PROPERTY FINAL sState : STRING(MAX_STRING_LENGTH)
GET
sState := TO_STRING(THIS^.eState);
END_GET
END_PROPERTY

END_FUNCTION_BLOCK

// ---- State Pattern Test/Test Subjects/Season State Pattern/FB_Winter.TcPOU
FUNCTION_BLOCK FB_Winter EXTENDS FB_SeasonBase
VAR
END_VAR

METHOD ChangeToWinterTyres
VAR_INPUT
END_VAR
THIS^._nTyresType := 0;
Tc2_System.ADSLOGSTR(msgCtrlMask := THIS^._nLogLevel,
                     msgFmtStr := 'Changed to winter tyres',
                     strArg := '');
END_METHOD

METHOD FB_init : BOOL
VAR_INPUT
    bInitRetains:           BOOL; // if TRUE, the retain variables are initialized (warm start / cold start)
    bInCopyCode:            BOOL;  // if TRUE, the instance afterwards gets moved into the copy code (online change)
    ipStateMachine:         I_StateMachine;
    ipParentObject:         I_Object;
END_VAR
THIS^._eState := E_Season.Winter;
END_METHOD

METHOD  NextSeason
VAR_INPUT
END_VAR
THIS^.ipStateMachine.SetState(THIS^.ipSeasonCtrl.StateSpring);
END_METHOD

METHOD OnEntry
VAR_INPUT
END_VAR
SUPER^.OnEntry();
THIS^._bWindBlowing     := FALSE;
THIS^._bRaining         := FALSE;
THIS^._bSunShining      := FALSE;
THIS^._bSnowing         := TRUE;
THIS^._nLeavesState     := 0;
END_METHOD

END_FUNCTION_BLOCK

// ---- State Pattern Test/Test Subjects/Season State Pattern/FB_Spring.TcPOU
FUNCTION_BLOCK FB_Spring EXTENDS FB_SeasonBase
VAR_INPUT
END_VAR
VAR_OUTPUT
END_VAR
VAR
END_VAR

METHOD ChangeToSummerTyres
VAR_INPUT
END_VAR
THIS^._nTyresType := 1;
Tc2_System.ADSLOGSTR(msgCtrlMask := THIS^._nLogLevel,
                     msgFmtStr := 'Changed to summer tyres',
                     strArg := '');
END_METHOD

METHOD FB_init : BOOL
VAR_INPUT
    bInitRetains:           BOOL; // if TRUE, the retain variables are initialized (warm start / cold start)
    bInCopyCode:            BOOL;  // if TRUE, the instance afterwards gets moved into the copy code (online change)
    ipStateMachine:         I_StateMachine;
    ipParentObject:         I_Object;
END_VAR
THIS^._eState := E_Season.Spring;
END_METHOD

METHOD  NextSeason
VAR_INPUT
END_VAR
THIS^.ipStateMachine.SetState(THIS^.ipSeasonCtrl.StateSummer);
END_METHOD

METHOD OnEntry
VAR_INPUT
END_VAR
SUPER^.OnEntry();
THIS^._bWindBlowing     := FALSE;
THIS^._bRaining         := TRUE;
THIS^._bSunShining      := FALSE;
THIS^._bSnowing         := TRUE;
THIS^._nLeavesState     := 1;
END_METHOD

METHOD OnExit
SUPER^.OnExit();
THIS^._bWindBlowing     := FALSE;
THIS^._bRaining         := FALSE;
THIS^._bSunShining      := FALSE;
THIS^._bSnowing         := TRUE;
THIS^._nLeavesState     := 1;
END_METHOD

END_FUNCTION_BLOCK

// ---- State Pattern Test/Test Subjects/Season State Pattern/FB_Summer.TcPOU
FUNCTION_BLOCK FB_Summer EXTENDS FB_SeasonBase
VAR_INPUT
END_VAR
VAR_OUTPUT
END_VAR
VAR
END_VAR

METHOD ChangeToSummerTyres
VAR_INPUT
END_VAR
THIS^._nTyresType := 1;
Tc2_System.ADSLOGSTR(msgCtrlMask := THIS^._nLogLevel,
                     msgFmtStr := 'Changed to summer tyres',
                     strArg := '');
END_METHOD

METHOD FB_init : BOOL
VAR_INPUT
    bInitRetains:           BOOL; // if TRUE, the retain variables are initialized (warm start / cold start)
    bInCopyCode:            BOOL;  // if TRUE, the instance afterwards gets moved into the copy code (online change)
    ipStateMachine:         I_StateMachine;
    ipParentObject:         I_Object;
END_VAR
THIS^._eState := E_Season.Summer;
END_METHOD

METHOD  NextSeason
VAR_INPUT
END_VAR
THIS^.ipStateMachine.SetState(THIS^.ipSeasonCtrl.StateAutumn);
END_METHOD

METHOD OnEntry
SUPER^.OnEntry();
THIS^._bWindBlowing     := FALSE;
THIS^._bRaining         := FALSE;
THIS^._bSunShining      := TRUE;
THIS^._bSnowing         := FALSE;
THIS^._nLeavesState     := 1;
END_METHOD

END_FUNCTION_BLOCK

// ---- State Pattern Test/Test Subjects/Season State Pattern/FB_Autumn.TcPOU
FUNCTION_BLOCK FB_Autumn EXTENDS FB_SeasonBase
VAR_INPUT
END_VAR
VAR_OUTPUT
END_VAR
VAR
END_VAR

METHOD FB_init : BOOL
VAR_INPUT
    bInitRetains:           BOOL; // if TRUE, the retain variables are initialized (warm start / cold start)
    bInCopyCode:            BOOL;  // if TRUE, the instance afterwards gets moved into the copy code (online change)
    ipStateMachine:         I_StateMachine;
    ipParentObject:         I_Object;
END_VAR
THIS^._eState := E_Season.Autumn;
END_METHOD

METHOD  NextSeason
VAR_INPUT
END_VAR
THIS^.ipStateMachine.SetState(THIS^.ipSeasonCtrl.StateWinter);
END_METHOD

METHOD OnEntry
VAR_INPUT
END_VAR
SUPER^.OnEntry();
THIS^._bWindBlowing     := TRUE;
THIS^._bRaining         := FALSE;
THIS^._bSunShining      := FALSE;
THIS^._bSnowing         := FALSE;
THIS^._nLeavesState     := 2;

Tc2_System.ADSLOGSTR(msgCtrlMask := THIS^._nLogLevel,
                     msgFmtStr := 'Leaves are changing color to yellow/orange/bright red',
                     strArg := '');
END_METHOD

METHOD OnExit
SUPER^.OnExit();
THIS^._bWindBlowing     := FALSE;
THIS^._bRaining         := FALSE;
THIS^._bSunShining      := FALSE;
THIS^._bSnowing         := FALSE;
THIS^._nLeavesState     := 2;
END_METHOD

END_FUNCTION_BLOCK

// ---- Action Test/FB_Action_Test.TcPOU
FUNCTION_BLOCK FB_Action_Test EXTENDS TcUnit.FB_TestSuite
VAR
END_VAR

TestActivateAction();
TestRunCyclicTaskAction();

METHOD PRIVATE TestActivateAction
VAR_INST
    fbObject: FB_ActionTestObject;
    fbActivate: FB_ActivateAction;
END_VAR
TcUnit.TEST('TestActivateTaskAction');

THIS^.AssertFalse(Condition := fbObject.bIsActivated,
                  Message := 'Object should not be activated yet');

fbActivate.Inputs(TRUE).Execute(fbObject);

THIS^.AssertTrue(Condition := fbObject.bIsActivated,
                 Message := 'Failed to activate object');

fbActivate.Inputs(FALSE).Execute(fbObject);

THIS^.AssertFalse(Condition := fbObject.bIsActivated,
                  Message := 'Failed to deactivate object');

TcUnit.TEST_FINISHED();
END_METHOD

METHOD PRIVATE TestRunCyclicTaskAction
VAR_INST
    nCyclesToRun: UDINT := 5;
    nCounter: UDINT := 0;
    fbObject: FB_ActionTestObject;
    fbRunCyclicTask: FB_RunCyclicTasksAction;
END_VAR
TcUnit.TEST('TestRunCyclicTaskAction');

fbRunCyclicTask.Execute(fbObject);
nCounter := nCounter + 1;

IF nCyclesToRun = nCounter THEN
    THIS^.AssertEquals_UDINT(Expected := nCyclesToRun,
                             Actual := fbObject.nCounter,
                             Message := 'Unexpected counter value of cyclic object');
    TcUnit.TEST_FINISHED();
END_IF
END_METHOD

END_FUNCTION_BLOCK
